	// Send Port
	ReconnectTimer		   : TON;
	ClientServerConnection : FB_ClientServerConnection;
	_ServerConnectionState : E_SocketConnectionState;
	SocketSend			   : FB_SocketSend;
	SendMessage			   : ST_TcpIpPayload;
	_Socket				   : T_HSOCKET;
	SendDelay			   : TON;
	PollTimer			   : TON;
	ResponseTimer		   : TON;
	SocketReceive		   : FB_SocketReceive;
	ReceiveMessage		   : ST_TcpIpPayload;

	//
	_ReconnectionTime : TIME := T#10S;
	_PollTime		  : TIME := T#100MS;
	_ReceiveTimeout	  : TIME := T#50S;
	_SendInterval	  : TIME := T#100MS;
END_VAR

VAR
	Commands		   : ARRAY[0..COMMAND_BUFFER] OF I_TcpIpSubscription;
	SendBuffer		   : ARRAY[0..COMMAND_BUFFER] OF ST_TcpIpPayload;
	PrioritySendBuffer : ARRAY[0..COMMAND_BUFFER] OF ST_TcpIpPayload;
END_VAR

VAR CONSTANT
	COMMAND_BUFFER : DINT := 99;
END_VAR

METHOD CyclicLogic
IF NOT _Initialized THEN
	Initialize();
	RETURN;
END_IF

SendReceiveSequence();
END_METHOD

METHOD Initialize
SocketCloseAll(sSrvNetId := '', bExecute := TRUE);
IF NOT SocketCloseAll.bBusy AND NOT SocketCloseAll.bError THEN
	_Initialized := TRUE;
END_IF
END_METHOD

{attribute 'monitoring' := 'call'}
PROPERTY Initialized : BOOL
GET
Initialized := _Initialized;
END_GET
SET
_Initialized := Initialized;
END_SET
END_PROPERTY

METHOD PROTECTED EvaluateResponse
VAR
	i : DINT;
END_VAR
FOR i := 0 TO COMMAND_BUFFER DO
	IF Commands[i] = 0 THEN
		EXIT;
	END_IF

	Commands[i].UpdateCommandResult(ADR(ReceiveMessage));
END_FOR

MEMSET(ADR(ReceiveMessage), 0, SIZEOF(ReceiveMessage));
END_METHOD

METHOD PROTECTED GetNextCommand
VAR
	i : DINT;
END_VAR
IF SendBuffer[0].Size <> 0 THEN
	MEMCPY(ADR(SendMessage), ADR(SendBuffer[0]), SIZEOF(SendBuffer[0]));
	FOR i := 0 TO (COMMAND_BUFFER - 1) DO
		MEMCPY(ADR(SendBuffer[i]), ADR(SendBuffer[i + 1]), SIZEOF(SendBuffer[i]));
	END_FOR
END_IF
END_METHOD

METHOD PROTECTED GetNextPriorityCommand
VAR
	i : DINT;
END_VAR
IF PrioritySendBuffer[0].Size <> 0 THEN
	MEMCPY(ADR(SendMessage), ADR(PrioritySendBuffer[0]), SIZEOF(PrioritySendBuffer[0]));
	FOR i := 0 TO (COMMAND_BUFFER - 1) DO
		MEMCPY(ADR(PrioritySendBuffer[i]), ADR(PrioritySendBuffer[i + 1]), SIZEOF(PrioritySendBuffer[i]));
	END_FOR
END_IF
END_METHOD

METHOD PROTECTED SendReceiveSequence
VAR_INST
	SequenceState : UDINT;
END_VAR
ClientServerConnection(sSrvNetID   := '',
					   sRemoteHost := _IP,
					   nRemotePort := _Port,
					   hSocket	   => _Socket,
					   eState	   => _ServerConnectionState);

SocketSend(sSrvNetId := '',
		   hSocket	 := _Socket,
		   cbLen	 := SendMessage.Size,
		   pSrc		 := ADR(SendMessage.Data),
		   tTimeout	 := T#5S);

SocketReceive(sSrvNetId := '',
			  hSocket	:= _Socket,
			  cbLen		:= SIZEOF(ReceiveMessage.Data),
			  pDest		:= ADR(ReceiveMessage.Data),
			  tTimeout	:= _ReceiveTimeout);

ReceiveMessage.Size := SIZEOF(ReceiveMessage.Data);

//
ReconnectTimer(PT := _ReconnectionTime);
PollTimer(PT := _PollTime);
ResponseTimer(PT := _ReceiveTimeout);
CASE SequenceState OF
	0:
		ClientServerConnection.bEnable := TRUE;
		IF _ServerConnectionState = eSOCKET_CONNECTED THEN
			SequenceState := SequenceState + 10;
		END_IF

		IF ClientServerConnection.bError THEN
			Trace.Error(_Name, CONCAT('ClientServerConnection.bError: ', TO_STRING(ClientServerConnection.nErrId)));
			SequenceState := 200;
		END_IF

	10:
		// SENDING -----------------------------------------------------------------------------------
		SendDelay(IN := NOT SendDelay.Q, PT := _SendInterval);
		IF SendMessage.Size = 0 THEN
			GetNextPriorityCommand();
		END_IF

		IF SendMessage.Size = 0 THEN
			GetNextCommand();
		END_IF

		IF SocketSend.bExecute AND NOT SocketSend.bBusy AND NOT SocketSend.bError THEN
			Trace.Info(_Name, 'Client sent');
			MEMSET(ADR(SendMessage), 0, SIZEOF(SendMessage));
			SocketSend.bExecute := FALSE;
		END_IF

		IF SendMessage.Size <> 0 AND NOT SocketSend.bExecute AND SendDelay.Q THEN
			SocketSend.bExecute := TRUE;
		END_IF

		IF SocketSend.bError THEN
			Trace.Error(_Name, CONCAT('SocketSend.bError: ', TO_STRING(SocketSend.nErrId)));
			SequenceState := 200;
		END_IF

		// RECEIVING -----------------------------------------------------------------------------------
		PollTimer.IN		   := TRUE;
		SocketReceive.bExecute := TRUE;
		IF PollTimer.Q AND NOT SocketReceive.bError AND NOT SocketReceive.bBusy THEN
			IF SocketReceive.nRecBytes > 0 THEN
				ResponseTimer.IN := FALSE;
				Trace.Info(_Name, 'Client recieved');
				EvaluateResponse();
			END_IF

			SequenceState := 11;
			// Stale connection, disconnected while socket was open
			IF SocketReceive.nRecBytes = 0 THEN
				ResponseTimer.IN := TRUE;
				IF ResponseTimer.Q THEN
					Trace.Error(_Name, 'Receive Connection stale - re-connect!');
					SequenceState := 200;
				END_IF
			END_IF
		END_IF

		IF SocketReceive.bError THEN
			Trace.Error(_Name, CONCAT('SocketReceive.bError: ', TO_STRING(SocketReceive.nErrId)));
			SequenceState := 200;
		END_IF

	11:
		PollTimer.IN		   := FALSE;
		SocketReceive.bExecute := FALSE;
		SequenceState		   := 10;

	200:
		ReconnectTimer.IN			   := TRUE;
		ResponseTimer.IN			   := FALSE;
		ClientServerConnection.bEnable := FALSE;
		SocketReceive.bExecute		   := FALSE;
		SocketSend.bExecute			   := FALSE;
		IF _ServerConnectionState = eSOCKET_DISCONNECTED AND ReconnectTimer.Q THEN
			ReconnectTimer.IN := FALSE;
			SequenceState	  := 0;
		END_IF
END_CASE
END_METHOD

{attribute 'monitoring' := 'call'}
PROPERTY ConnectionState : E_SocketConnectionState
GET
ConnectionState := _ServerConnectionState;
END_GET
END_PROPERTY

{attribute 'monitoring' := 'call'}
PROPERTY IP : T_IPv4Addr
SET
_IP := IP;
END_SET
END_PROPERTY

{attribute 'monitoring' := 'call'}
PROPERTY PollTime : TIME
SET
_PollTime := PollTime;
END_SET
END_PROPERTY

{attribute 'monitoring' := 'call'}
PROPERTY Port : UDINT
SET
_Port := Port;
END_SET
END_PROPERTY

{attribute 'monitoring' := 'call'}
PROPERTY ReceiveTimeout : TIME
SET
_ReceiveTimeout := ReceiveTimeout;
END_SET
END_PROPERTY

{attribute 'monitoring' := 'call'}
PROPERTY ReconnectionTime : TIME
SET
_ReconnectionTime := ReconnectionTime;
END_SET
END_PROPERTY

METHOD RegisterCommand
VAR_INPUT
	Command : I_TcpIpSubscription;
END_VAR

VAR
	i : DINT;
END_VAR
FOR i := 0 TO COMMAND_BUFFER DO
	IF Commands[i] = 0 THEN
		Commands[i] := Command;
		RETURN;
	END_IF
END_FOR
END_METHOD

METHOD SendCommand
VAR_INPUT
	Command : POINTER TO ST_TcpIpPayload;
END_VAR

VAR
	i : DINT;
END_VAR
FOR i := 0 TO COMMAND_BUFFER DO
	IF SendBuffer[i].Size = 0 THEN
		MEMCPY(ADR(SendBuffer[i]), Command, SIZEOF(SendBuffer[i]));
		RETURN;
	END_IF
END_FOR
END_METHOD

{attribute 'monitoring' := 'call'}
PROPERTY SendInterval : TIME
SET
_SendInterval := SendInterval;
END_SET
END_PROPERTY

METHOD SendPriorityCommand
VAR_INPUT
	Command : POINTER TO ST_TcpIpPayload;
END_VAR

VAR
	i : DINT;
END_VAR
FOR i := 0 TO COMMAND_BUFFER DO
	IF PrioritySendBuffer[i].Size = 0 THEN
		MEMCPY(ADR(PrioritySendBuffer[i]), Command, SIZEOF(PrioritySendBuffer[i]));
		RETURN;
	END_IF
END_FOR
END_METHOD

PROPERTY Socket : T_HSOCKET
GET
Socket := _Socket;
END_GET
END_PROPERTY

END_FUNCTION_BLOCK

// HMI/Interface/I_Button
INTERFACE I_Button EXTENDS I_Base

{attribute 'monitoring' := 'call'}
PROPERTY Active : BOOL
GET
END_GET
END_PROPERTY

{attribute 'monitoring' := 'call'}
PROPERTY Name : STRING
GET
END_GET
SET
END_SET
END_PROPERTY

PROPERTY Permissive : I_Permissive
GET
END_GET
END_PROPERTY

END_INTERFACE

// HMI/Interface/I_StringCollection
INTERFACE I_StringCollection

METHOD AddString
VAR_INPUT
	StringToAdd : T_MaxString;
END_VAR
END_METHOD

METHOD Clear : BOOL
VAR_INPUT
END_VAR
END_METHOD

PROPERTY Entries : UDINT
GET
END_GET
END_PROPERTY

END_INTERFACE

// HMI/Button
FUNCTION_BLOCK Button IMPLEMENTS I_Button
VAR
	_Name		: STRING;
	_Active		: BOOL;
	_Permissive : PermissiveInterlock;
END_VAR

{attribute 'monitoring' := 'call'}
PROPERTY Active : BOOL
GET
Active := _Active;
END_GET
END_PROPERTY

{attribute 'monitoring' := 'call'}
PROPERTY Name : STRING
GET
Name := _Name;
END_GET
SET
_Name := Name;
END_SET
END_PROPERTY

PROPERTY Permissive : I_Permissive
GET
Permissive := _Permissive;
END_GET
END_PROPERTY

END_FUNCTION_BLOCK

// Permissive Interlock/PermissiveInterlock
FUNCTION_BLOCK PermissiveInterlock IMPLEMENTS I_Permissive
VAR
	_OK				 : BOOL				   := TRUE;
	Permissive		 : ARRAY[0..9] OF BOOL := [TRUE, TRUE, TRUE, TRUE, TRUE, TRUE, TRUE, TRUE, TRUE, TRUE];
	PermissiveReason : ARRAY[0..9] OF STRING;
END_VAR

METHOD PROTECTED Check : BOOL
VAR
	i : UDINT;
END_VAR
_OK := TRUE;
FOR i := 0 TO 9 DO
	IF NOT Permissive[i] THEN
		_OK := FALSE;
	END_IF
END_FOR
END_METHOD

{attribute 'monitoring' := 'call'}
PROPERTY OK : BOOL
GET
OK := _OK;
END_GET
END_PROPERTY

METHOD Set
VAR_INPUT
	Index  : UDINT(0..9);
	Reason : STRING;
	Value  : BOOL;
END_VAR
Permissive[Index]		:= Value;
PermissiveReason[Index] := Reason;
Check();
END_METHOD

END_FUNCTION_BLOCK

// Kinematic Group/Interface/I_KinematicGroup
INTERFACE I_KinematicGroup EXTENDS I_Component, I_Override, I_TaskResult, I_Resettable

METHOD AddAcsAxis : BOOL
VAR_INPUT
	AxisId : UDINT;
END_VAR
END_METHOD

METHOD AddMcsAxis : BOOL
VAR_INPUT
	AxisId : UDINT;
END_VAR
END_METHOD

METHOD BuildGroup
VAR_INPUT
END_VAR
END_METHOD

METHOD DissolveGroup
VAR_INPUT
END_VAR
END_METHOD

{attribute 'monitoring' := 'call'}
PROPERTY Status : E_KinStatus
GET
END_GET
END_PROPERTY

END_INTERFACE

// Kinematic Group/KinematicGroup
FUNCTION_BLOCK KinematicGroup EXTENDS CyclicComponent IMPLEMENTS I_KinematicGroup, I_Initializable
VAR
	NcToPlc AT %I* : NCTOPLC_NCICHANNEL_REF;
	PlcToNc AT %Q* : PLCTONC_NCICHANNEL_REF;
	KinAxes		   : ST_KinAxes;
	KinConfigGroup : FB_KinConfigGroup;
	KinResetGroup  : FB_KinResetGroup;
	{attribute 'hide'}
	_Initialized : BOOL;
	{attribute 'hide'}
	_Busy : BOOL;
	{attribute 'hide'}
	_Error : BOOL;
	{attribute 'hide'}
	_ErrorId : UDINT;
END_VAR

METHOD DeregisterWithParent
VAR_INPUT
	Parent : I_ContainComponents;
END_VAR
SUPER^.DeregisterWithParent(Parent);
Parent.DeregisterInitialize(THIS^);
END_METHOD

METHOD RegisterWithParent
VAR_INPUT
	Parent : I_ContainComponents;
END_VAR
SUPER^.RegisterWithParent(Parent);
Parent.RegisterInitialize(THIS^);
END_METHOD

METHOD CyclicLogic
IF NOT Initialized THEN
	Initialize();
	RETURN;
END_IF

//
KinConfigGroup(stAxesList := KinAxes, stKinRefIn := NcToPlc);
IF KinConfigGroup.bError THEN
	_Error	 := TRUE;
	_ErrorId := KinConfigGroup.nErrorId;
END_IF

KinConfigGroup.bExecute := FALSE;

//
KinResetGroup(nItpChannelId := NcToPlc.ChnId, stKinRefIn := NcToPlc, stAxesList := KinAxes);
IF KinResetGroup.bError THEN
	_Error	 := TRUE;
	_ErrorId := KinResetGroup.nErrorId;
END_IF

KinResetGroup.bExecute := FALSE;

//
_Busy := KinConfigGroup.bBusy;
END_METHOD

METHOD Initialize
VAR
	i : DINT;
END_VAR
IF NOT Initialized THEN
	IF KinAxes.nAxisIdsAcs[1] = 0 THEN
		Trace.LogMessage(Name, 'Init failed - at least one ACS Axis needs to be added to Kinematic!');
		RETURN;
	END_IF

	IF KinAxes.nAxisIdsMcs[1] = 0 THEN
		Trace.LogMessage(Name, 'Init failed - at least one MCS Axis needs to be added to Kinematic!');
		RETURN;
	END_IF

	IF F_GetMappingStatus(ADR(NcToPlc), SIZEOF(NcToPlc)) <> EPlcMappingStatus.MS_Mapped THEN
		Trace.LogMessage(Name, 'Init failed - NcToPlc not mapped to Kinematic Channel!');
		RETURN;
	END_IF

	IF F_GetMappingStatus(ADR(PlcToNc), SIZEOF(PlcToNc)) <> EPlcMappingStatus.MS_Mapped THEN
		Trace.LogMessage(Name, 'Init failed - PlcToNc not mapped to Kinematic Channel!');
		RETURN;
	END_IF

	Initialized := TRUE;
END_IF
END_METHOD

{attribute 'monitoring' := 'call'}
PROPERTY Initialized : BOOL
GET
Initialized := _Initialized;
END_GET
SET
_Initialized := Initialized;
END_SET
END_PROPERTY

METHOD AddAcsAxis : BOOL
VAR_INPUT
	AxisId : UDINT;
END_VAR

VAR
	i : DINT;
END_VAR
IF AxisId = 0 THEN
	RETURN;
END_IF

FOR i := 1 TO 8 DO
	IF KinAxes.nAxisIdsAcs[i] = 0 THEN
		KinAxes.nAxisIdsAcs[i] := AxisId;
		AddAcsAxis			   := TRUE;
		RETURN;
	END_IF
END_FOR
END_METHOD

METHOD AddMcsAxis : BOOL
VAR_INPUT
	AxisId : UDINT;
END_VAR

VAR
	i : DINT;
END_VAR
IF AxisId = 0 THEN
	RETURN;
END_IF

FOR i := 1 TO 8 DO
	IF KinAxes.nAxisIdsMcs[i] = 0 THEN
		KinAxes.nAxisIdsMcs[i] := AxisId;
		AddMcsAxis			   := TRUE;
		RETURN;
	END_IF
END_FOR
END_METHOD

METHOD BuildGroup
VAR_INPUT
END_VAR
IF Busy THEN
	RETURN;
END_IF

KinConfigGroup.bCartesianMode := TRUE;
KinConfigGroup.bExecute		  := TRUE;
END_METHOD

METHOD DissolveGroup
VAR_INPUT
END_VAR
IF Busy THEN
	RETURN;
END_IF

KinConfigGroup.bCartesianMode := FALSE;
KinConfigGroup.bExecute		  := TRUE;
END_METHOD

{attribute 'monitoring' := 'call'}
PROPERTY Override : LREAL
SET
PlcToNc.ChnAxesOvr	  := TO_UDINT(Override * 10_000);
PlcToNc.ChnSpindleOvr := TO_UDINT(Override * 10_000);
END_SET
END_PROPERTY

{attribute 'monitoring' := 'call'}
PROPERTY Status : E_KinStatus
GET
Status := F_KinGetChnOperationState(NcToPlc);
END_GET
END_PROPERTY

METHOD Reset
_Error				   := FALSE;
_ErrorId			   := 0;
KinResetGroup.bExecute := TRUE;
END_METHOD

{attribute 'monitoring' := 'call'}
PROPERTY Busy : BOOL
GET
Busy := _Busy;
END_GET
END_PROPERTY

{attribute 'monitoring' := 'call'}
PROPERTY Error : BOOL
GET
Error := _Error;
END_GET
END_PROPERTY

{attribute 'monitoring' := 'call'}
PROPERTY ErrorId : UDINT
GET
ErrorId := _ErrorId;
END_GET
END_PROPERTY

END_FUNCTION_BLOCK

// Kinematic Group/KinematicGroup_TcEvents
FUNCTION_BLOCK KinematicGroup_TcEvents EXTENDS CyclicComponent IMPLEMENTS I_EventReactionTcEvents
VAR
	KinematicGroup : I_KinematicGroup;
	Events		   : TcEventClass('Kinematic Group Events');
END_VAR

METHOD GetHighestActiveEventReaction : DINT
GetHighestActiveEventReaction := Events.GetHighestActiveEventReaction();
END_METHOD

METHOD GetHighestActiveEventSeverity : TcEventSeverity
GetHighestActiveEventSeverity := Events.GetHighestActiveEventSeverity();
END_METHOD

METHOD Reset
Events.Reset();
END_METHOD

METHOD SetEventReactions
VAR_INPUT
	Verbose	 : DINT := 0;
	Info	 : DINT := 1;
	Warning	 : DINT := 2;
	Error	 : DINT := 3;
	Critical : DINT := 4;
END_VAR
Events.SetEventReactions(Verbose,
						 Info,
						 Warning,
						 Error,
						 Critical);
END_METHOD

METHOD CyclicLogic
IF KinematicGroup = 0 THEN
	RETURN;
END_IF

IF KinematicGroup.Error THEN
	Events.Arguments(E_KinematicGroup.KinematicGroupError).Clear().AddString(TO_STRING(KinematicGroup.ErrorId));
	Events.RaiseEvent(E_KinematicGroup.KinematicGroupError);
END_IF
END_METHOD

(*FB_Init is always available implicitly and it is used primarily for initialization.
The return value is not evaluated. For a specific influence, you can also declare the
methods explicitly and provide additional code there with the standard initialization
code. You can evaluate the return value.*)
METHOD FB_Init : BOOL
VAR_INPUT
	(* TRUE: the retain variables are initialized (reset warm / reset cold)*)
	bInitRetains : BOOL;

	(* TRUE: the instance will be copied to the copy code afterward (online change)   *)
	bInCopyCode	   : BOOL;
	Name		   : T_MaxString;
	KinematicGroup : I_KinematicGroup;
END_VAR
THIS^.KinematicGroup := KinematicGroup;
Events.GenerateTcEvents(KinematicGroup.Name, ADR(TC_Events.KinematicGroup), SIZEOF(ST_KinematicGroup));
END_METHOD

END_FUNCTION_BLOCK

// Modes/PackMLModeControl
FUNCTION_BLOCK PackMLModeControl IMPLEMENTS I_Mode, I_Cyclic
VAR
	{attribute 'hide'}
	_CurrentMode : DINT;
	{attribute 'hide'}
	ModeManager	  : FB_PMLUnitModeManager;
	ModeCommand	  : DINT;
	_StateMachine : I_Statemachine;
END_VAR

METHOD ChangeMode
VAR_INPUT
	RequestedMode : DINT;
END_VAR
IF RequestedMode <= 0 OR RequestedMode > 31 THEN
	Trace.LogMessage('PackML Mode Controller', ' - Requested Mode is not valid 1..31');
	RETURN;
END_IF

ModeCommand := RequestedMode;
END_METHOD

{attribute 'monitoring' := 'call'}
PROPERTY CurrentMode : DINT
GET
CurrentMode := _CurrentMode;
END_GET
END_PROPERTY

METHOD CyclicLogic
VAR_INST
	LastModeCommand		: DINT;
	ModeChangeRequested : BOOL;
END_VAR
IF _CurrentMode = 0 THEN
	ModeChangeRequested := TRUE;
	ModeCommand			:= E_PMLProtectedUnitMode.Production;
	LastModeCommand		:= ModeCommand;
ELSIF ModeCommand <> LastModeCommand THEN
	ModeChangeRequested := TRUE;
	LastModeCommand		:= ModeCommand;
END_IF

IF ModeChangeRequested THEN
	{warning disable C0196}
	ModeManager(bExecute	 := TRUE,
				eModeCommand := ModeCommand,
				eState		 := _StateMachine.CurrentState,
				eModeStatus	 => _CurrentMode);

	IF ModeManager.bDone THEN
		ModeManager(bExecute := FALSE);
		ModeChangeRequested := FALSE;
	ELSIF ModeManager.bError THEN
		IF ModeManager.nErrorId = 1 THEN
			Trace.LogMessage('PackML Mode Controller', 'Requested mode is not defined or Mode change is disabled in this PackML state!');
		ELSE
			Trace.LogMessage('PackML Mode Controller', 'Mode change error, check PackML configuration!');
		END_IF

		ModeManager(bExecute := FALSE);
		_StateMachine.ChangeState(TO_UDINT(E_PMLCommand.Abort));
		ModeCommand			:= E_PMLProtectedUnitMode.Production;
		ModeChangeRequested := FALSE;
	END_IF
END_IF
END_METHOD

PROPERTY StateMachine : I_StateMachine
SET
_StateMachine := StateMachine;
END_SET
END_PROPERTY

END_FUNCTION_BLOCK

// Module PackML/PackMLModule
FUNCTION_BLOCK ABSTRACT PackMLModule EXTENDS Module IMPLEMENTS I_Module, I_ContainStatemachine
VAR
	_Statemachine : PackMLStatemachine_ModuleIntegrated('Statemachine');
	SequenceState : UDINT;
END_VAR

(*FB_Init is always available implicitly and it is used primarily for initialization.
The return value is not evaluated. For a specific influence, you can also declare the
methods explicitly and provide additional code there with the standard initialization
code. You can evaluate the return value.*)
METHOD FB_Init : BOOL
VAR_INPUT
	(* TRUE: the retain variables are initialized (reset warm / reset cold)*)
	bInitRetains	: BOOL;
	(* TRUE: the instance will be copied to the copy code afterward (online change)   *)
	bInCopyCode	: BOOL;
	Name	: T_MaxString;
END_VAR
_Statemachine.RegisterWithParent(THIS^);
END_METHOD

METHOD Aborted : BOOL;
Aborted := TRUE;
END_METHOD

METHOD Aborting : BOOL
Aborting := TRUE;
END_METHOD

METHOD Clearing : BOOL
Clearing := TRUE;
END_METHOD

METHOD Completed : BOOL
Completed := TRUE;
END_METHOD

METHOD Completing : BOOL
Completing := TRUE;
END_METHOD

METHOD Execute : BOOL
Execute := TRUE;
END_METHOD

METHOD Held : BOOL
Held := TRUE;
END_METHOD

METHOD Holding : BOOL
Holding := TRUE;
END_METHOD

METHOD Idle : BOOL
Idle := TRUE;
END_METHOD

METHOD Resetting : BOOL
Resetting := TRUE;
END_METHOD

METHOD Starting : BOOL
Starting := TRUE;
END_METHOD

METHOD Stopped : BOOL
Stopped := TRUE;
END_METHOD

METHOD Stopping : BOOL
Stopping := TRUE;
END_METHOD

METHOD Suspended : BOOL
Suspended := TRUE;
END_METHOD

METHOD Suspending : BOOL
Suspending := TRUE;
END_METHOD

METHOD Unholding : BOOL
Unholding := TRUE;
END_METHOD

METHOD Unsuspending : BOOL
Unsuspending := TRUE;
END_METHOD

METHOD CyclicLogic
StateSelect();
SUPER^.CyclicLogic();
END_METHOD

PROPERTY Statemachine : I_Statemachine
GET
Statemachine := _Statemachine;
END_GET
END_PROPERTY

METHOD PRIVATE StateSelect
VAR_INST
	ClearingTon : TON;
	LastState	: DINT;
END_VAR
IF LastState <> _Statemachine.CurrentState THEN
	SequenceState := 0;
	LastState	  := _Statemachine.CurrentState;
END_IF

CASE _Statemachine.CurrentState OF
	E_PMLState.Undefined:
		;

	E_PMLState.Clearing:
		ClearingTon(IN := TRUE, PT := ApplicationBaseParameter.ClearingTimeout);
		IF Clearing() THEN
			ClearingTon(IN := FALSE);
			_Statemachine.StateComplete();
		END_IF

		IF ClearingTon.Q THEN
			ClearingTon(IN := FALSE);
			Trace.LogMessage('Clearing Timeout exeeded! - ', _Name);
			_Statemachine.ChangeState(E_PMLCommand.Abort);
		END_IF

	E_PMLState.Stopped:
		Stopped();

	E_PMLState.Starting:
		IF Starting() THEN
			_Statemachine.StateComplete();
		END_IF

	E_PMLState.Idle:
		Idle();

	E_PMLState.Suspended:
		Suspended();

	E_PMLState.Execute:
		Execute();

	E_PMLState.Stopping:
		IF Stopping() THEN
			_Statemachine.StateComplete();
		END_IF

	E_PMLState.Aborting:
		IF Aborting() THEN
			_Statemachine.StateComplete();
		END_IF

	E_PMLState.Aborted:
		Aborted();

	E_PMLState.Holding:
		IF Holding() THEN
			_Statemachine.StateComplete();
		END_IF

	E_PMLState.Held:
		Held();

	E_PMLState.Unholding:
		IF Unholding() THEN
			_Statemachine.StateComplete();
		END_IF

	E_PMLState.Suspending:
		IF Suspending() THEN
			_Statemachine.StateComplete();
		END_IF

	E_PMLState.Unsuspending:
		IF Unsuspending() THEN
			_Statemachine.StateComplete();
		END_IF

	E_PMLState.Resetting:
		IF Resetting() THEN
			_Statemachine.StateComplete();
		END_IF

	E_PMLState.Completing:
		IF Completing() THEN
			_Statemachine.StateComplete();
		END_IF

	E_PMLState.Completed:
		Completed();
END_CASE
END_METHOD

END_FUNCTION_BLOCK

// Statemachine/Interface/I_ContainStatemachine
INTERFACE I_ContainStatemachine EXTENDS I_Base

PROPERTY Statemachine : I_Statemachine
GET
END_GET
END_PROPERTY

END_INTERFACE

// Statemachine/PackML/PackMLStatemachine_ModuleIntegrated
FUNCTION_BLOCK PackMLStatemachine_ModuleIntegrated EXTENDS CyclicComponent IMPLEMENTS I_StateMachine
VAR
	StateMachine   : FB_PMLStateMachine;
	StateCommand   : E_PMLCommand;
	_CurrentState  : E_PMLState;
	ModeController : PackMLModeControl := (StateMachine := THIS^);
END_VAR

PROPERTY Mode : I_Mode
GET
Mode := ModeController;
END_GET
SET
// Fix defined in PackML
END_SET
END_PROPERTY

METHOD ChangeState
VAR_INPUT
	StateCommand : DINT;
END_VAR
IF StateCommand <= 0 OR StateCommand > 17 THEN
	Trace.LogMessage('PackML Statemachine ChangeState()', 'StateId is not a PackML State');
END_IF

{warning disable C0196}
THIS^.StateCommand := StateCommand;
END_METHOD

{attribute 'monitoring' := 'call'}
PROPERTY CurrentState : DINT
GET
CurrentState := _CurrentState;
END_GET
END_PROPERTY

METHOD CyclicLogic
VAR_INST
	ClearingTon : TON;
END_VAR
ModeController.CyclicLogic();
IF _CurrentState = E_PMLState.Undefined AND Mode.CurrentMode <> 0 THEN
	StateCommand := E_PMLCommand.Abort;
END_IF

StateMachine(eMode			  := TO_DINT(Mode.CurrentMode),
			 eCommand		  := StateCommand,
			 stSubUnitInfoRef :=,
			 stOptions		  :=,
			 eState			  => _CurrentState,
			 sState			  =>,
			 bError			  =>,
			 nErrorID		  =>);

CASE _CurrentState OF
	E_PMLState.Clearing:
		ClearingTon(IN := TRUE, PT := ApplicationBaseParameter.ClearingTimeout);
		IF ClearingTon.Q THEN
			ClearingTon(IN := FALSE);
			Trace.LogMessage('Clearing Timeout exeeded!', 'ApplicationBaseParameter.ClearingTimeout');
			StateCommand := E_PMLCommand.Abort;
		END_IF

ELSE
	ClearingTon(IN := FALSE);
END_CASE
END_METHOD

METHOD StateComplete
StateMachine.M_StateComplete();
END_METHOD

{attribute 'hide'} 
PROPERTY States : I_StateList
GET
States := 0;
END_GET
END_PROPERTY

END_FUNCTION_BLOCK

// Motion/Interface/I_Axis_PTP
INTERFACE I_Axis_PTP EXTENDS I_Axis, I_AxisMoveAbsolute, I_AxisMoveModulo, I_AxisMoveRelative, I_AxisMoveVelocity

END_INTERFACE

// Motion/Interface/I_AxisMoveAbsolute
INTERFACE I_AxisMoveAbsolute EXTENDS I_Base

METHOD MoveAbsolute
VAR_INPUT
	TargetPosition : LREAL;
	AbortPrevious  : BOOL := TRUE;
END_VAR
END_METHOD

END_INTERFACE

// Motion/Interface/I_AxisMoveModulo
INTERFACE I_AxisMoveModulo EXTENDS I_Base

METHOD MoveModulo : BOOL
VAR_INPUT
	Position	  : LREAL;
	Direction	  : MC_Direction := MC_Direction.MC_Shortest_Way;
	AbortPrevious : BOOL		 := TRUE;
END_VAR
END_METHOD

END_INTERFACE

// Motion/Interface/I_AxisMoveRelative
INTERFACE I_AxisMoveRelative EXTENDS I_Base

METHOD MoveRelative : BOOL
VAR_INPUT
	Distance	  : LREAL;
	AbortPrevious : BOOL := TRUE;
END_VAR
END_METHOD

END_INTERFACE

// Motion/Interface/I_AxisMoveVelocity
INTERFACE I_AxisMoveVelocity EXTENDS I_Base

METHOD MoveVelocity : BOOL
VAR_INPUT
	Velocity	  : LREAL;
	AbortPrevious : BOOL := TRUE;
END_VAR
END_METHOD

END_INTERFACE

// Motion/Interface/I_AxisGear
INTERFACE I_AxisGear EXTENDS I_Base

METHOD GearIn
VAR_INPUT
END_VAR
END_METHOD

PROPERTY GearInMultiMasterOptions : ST_GearInMultiMasterOptions
SET
END_SET
END_PROPERTY

METHOD GearOut
VAR_INPUT
END_VAR
END_METHOD

{attribute 'monitoring' := 'call'}
PROPERTY GearRatioMaster1 : LREAL
SET
END_SET
END_PROPERTY

{attribute 'monitoring' := 'call'}
PROPERTY GearRatioMaster2 : LREAL
SET
END_SET
END_PROPERTY

{attribute 'monitoring' := 'call'}
PROPERTY GearRatioMaster3 : LREAL
SET
END_SET
END_PROPERTY

{attribute 'monitoring' := 'call'}
PROPERTY GearRatioMaster4 : LREAL
SET
END_SET
END_PROPERTY

PROPERTY Master1 : I_Axis
SET
END_SET
END_PROPERTY

PROPERTY Master2 : I_Axis
SET
END_SET
END_PROPERTY

PROPERTY Master3 : I_Axis
SET
END_SET
END_PROPERTY

PROPERTY Master4 : I_Axis
SET
END_SET
END_PROPERTY

END_INTERFACE

// Motion/Interface/I_SlaveAxis
INTERFACE I_SlaveAxis EXTENDS I_Axis_PTP, I_AxisGear

END_INTERFACE

// Motion/Axis_TcEvents
FUNCTION_BLOCK Axis_TcEvents EXTENDS CyclicComponent IMPLEMENTS I_EventReactionTcEvents
VAR
	Axis   : I_Axis;
	Events : TcEventClass(CONCAT(Name, ' Events'));
END_VAR

METHOD GetHighestActiveEventReaction : DINT
GetHighestActiveEventReaction := Events.GetHighestActiveEventReaction();
END_METHOD

METHOD GetHighestActiveEventSeverity : TcEventSeverity
GetHighestActiveEventSeverity := Events.GetHighestActiveEventSeverity();
END_METHOD

METHOD Reset
Events.Reset();
END_METHOD

METHOD SetEventReactions
VAR_INPUT
	Verbose	 : DINT := 0;
	Info	 : DINT := 1;
	Warning	 : DINT := 2;
	Error	 : DINT := 3;
	Critical : DINT := 4;
END_VAR
Events.SetEventReactions(Verbose,
						 Info,
						 Warning,
						 Error,
						 Critical);
END_METHOD

METHOD CyclicLogic
IF Axis.MotionTasks.Error THEN
	Events.Arguments(E_Nc2Axis.AxisError).Clear().AddString(Axis.MotionTasks.ErrorTask).AddString(TO_STRING(Axis.MotionTasks.ErrorId));
	Events.RaiseEvent(E_Nc2Axis.AxisError);
END_IF
END_METHOD

(*FB_Init is always available implicitly and it is used primarily for initialization.
The return value is not evaluated. For a specific influence, you can also declare the
methods explicitly and provide additional code there with the standard initialization
code. You can evaluate the return value.*)
METHOD FB_Init : BOOL
VAR_INPUT
	(* TRUE: the retain variables are initialized (reset warm / reset cold)*)
	bInitRetains : BOOL;

	(* TRUE: the instance will be copied to the copy code afterward (online change)   *)
	bInCopyCode : BOOL;
	Name		: T_MaxString;
	Axis		: I_Axis;
END_VAR
THIS^.Axis := Axis;
Events.GenerateTcEvents(Axis.Name, ADR(TC_events.Nc2Axis), SIZEOF(ST_Nc2Axis));
END_METHOD

END_FUNCTION_BLOCK

// Motion/AxisPTP
FUNCTION_BLOCK AxisPTP EXTENDS Axis IMPLEMENTS I_Axis_PTP
VAR
	// Tasks
	{attribute 'hide'}
	MoveAbsoluteTask : MoveAbsoluteTask := (Name := 'MC Move Absolute');
	{attribute 'hide'}
	MoveRelativeTask : MoveRelativeTask := (Name := 'MC Move Relative');
	{attribute 'hide'}
	MoveModuloTask : MoveModuloTask := (Name := 'MC Move Modulo');
	{attribute 'hide'}
	MoveVelocityTask : MoveVelocityTask := (Name := 'MC Move Velocity');
END_VAR

(*FB_Init is always available implicitly and it is used primarily for initialization.
The return value is not evaluated. For a specific influence, you can also declare the
methods explicitly and provide additional code there with the standard initialization
code. You can evaluate the return value.*)
METHOD FB_Init : BOOL
VAR_INPUT
	(* TRUE: the retain variables are initialized (reset warm / reset cold)*)
	bInitRetains : BOOL;

	(* TRUE: the instance will be copied to the copy code afterward (online change)   *)
	bInCopyCode : BOOL;
	Name		: T_MaxString;
	Axis		: REFERENCE TO AXIS_REF;
END_VAR
// Register all Motion Tasks to Collection
MotionTaskCollection.AddTask(MoveAbsoluteTask);
MotionTaskCollection.AddTask(MoveRelativeTask);
MotionTaskCollection.AddTask(MoveModuloTask);
MotionTaskCollection.AddTask(MoveVelocityTask);
END_METHOD

METHOD MoveAbsolute
VAR_INPUT
	TargetPosition : LREAL;
	AbortPrevious  : BOOL := TRUE;
END_VAR
IF Error THEN
	RETURN;
ELSE
	IF Busy AND NOT AbortPrevious THEN
		RETURN;
	END_IF
END_IF

MoveAbsoluteTask.BufferMode		:= _McBufferMode;
MoveAbsoluteTask.MoveOptions	:= _MoveOptions;
MoveAbsoluteTask.TargetPosition := TargetPosition;
MoveAbsoluteTask.Execute();
END_METHOD

METHOD MoveModulo : BOOL
VAR_INPUT
	Position	: LREAL;
	Direction	: MC_Direction := .MC_Direction.MC_Shortest_Way;
	AbortPrevious	: BOOL := TRUE;
END_VAR
IF Error THEN
	RETURN;
ELSE
	IF Busy AND NOT AbortPrevious THEN
		RETURN;
	END_IF
END_IF

MoveModuloTask.BufferMode	  := _McBufferMode;
MoveModuloTask.MoveOptions	  := _MoveOptions;
MoveModuloTask.Direction	  := Direction;
MoveModuloTask.TargetPosition := Position;
MoveModuloTask.Execute();
END_METHOD

METHOD MoveRelative : BOOL
VAR_INPUT
	Distance	  : LREAL;
	AbortPrevious : BOOL := TRUE;
END_VAR
IF Error THEN
	RETURN;
ELSE
	IF Busy AND NOT AbortPrevious THEN
		RETURN;
	END_IF
END_IF

MoveRelativeTask.BufferMode		:= _McBufferMode;
MoveRelativeTask.MoveOptions	:= _MoveOptions;
MoveRelativeTask.TargetDistance := Distance;
MoveRelativeTask.Execute();
END_METHOD

METHOD MoveVelocity : BOOL
VAR_INPUT
	Velocity	  : LREAL;
	AbortPrevious : BOOL := TRUE;
END_VAR
IF Error THEN
	RETURN;
ELSE
	IF Busy AND NOT AbortPrevious THEN
		RETURN;
	END_IF
END_IF

MoveVelocityTask.BufferMode		:= _McBufferMode;
MoveVelocityTask.MoveOptions	:= _MoveOptions;
MoveVelocityTask.TargetVelocity := Velocity;
MoveVelocityTask.Execute();
END_METHOD

END_FUNCTION_BLOCK

// Motion/AxisPTP_HMI
FUNCTION_BLOCK AxisPTP_HMI EXTENDS HmiFunction
VAR
	Axis : I_Axis_PTP;
	{ attribute 'TcHmiSymbol.AddSymbol' }
	{ attribute 'TcHmiSymbol.AddSymbol.UserGroups' := '__SystemAdministrators,Admin' }
	AxisPTP_HMI : ST_AxisPTP_HMI;
END_VAR

PROPERTY DisablePermissive : I_Permissive
GET
DisablePermissive := AxisPTP_HMI.Disable.Permissive;
END_GET
END_PROPERTY

PROPERTY EnablePermissive : I_Permissive
GET
EnablePermissive := AxisPTP_HMI.Enable.Permissive;
END_GET
END_PROPERTY

PROPERTY HomePermissive : I_Permissive
GET
HomePermissive := AxisPTP_HMI.Home.Permissive;
END_GET
END_PROPERTY

PROPERTY JogBackwardFastPermissive : I_Permissive
GET
JogBackwardFastPermissive := AxisPTP_HMI.JogBackwardFast.Permissive;
END_GET
END_PROPERTY

PROPERTY JogBackwardSlowPermissive : I_Permissive
GET
JogBackwardSlowPermissive := AxisPTP_HMI.JogBackwardSlow.Permissive;
END_GET
END_PROPERTY

PROPERTY JogForwardFastPermissive : I_Permissive
GET
JogForwardFastPermissive := AxisPTP_HMI.JogForwardFast.Permissive;
END_GET
END_PROPERTY

PROPERTY JogForwardSlowPermissive : I_Permissive
GET
JogForwardSlowPermissive := AxisPTP_HMI.JogForwardSlow.Permissive;
END_GET
END_PROPERTY

PROPERTY MoveAbsolutePermissive : I_Permissive
GET
MoveAbsolutePermissive := AxisPTP_HMI.MoveAbsolute.Permissive;
END_GET
END_PROPERTY

PROPERTY MoveModuloPermissive : I_Permissive
GET
MoveModuloPermissive := AxisPTP_HMI.MoveModulo.Permissive;
END_GET
END_PROPERTY

PROPERTY MoveRelativePermissive : I_Permissive
GET
MoveRelativePermissive := AxisPTP_HMI.MoveRelative.Permissive;
END_GET
END_PROPERTY

PROPERTY MoveVelocityPermissive : I_Permissive
GET
MoveVelocityPermissive := AxisPTP_HMI.MoveVelocity.Permissive;
END_GET
END_PROPERTY

PROPERTY ResetPermissive : I_Permissive
GET
ResetPermissive := AxisPTP_HMI.Reset.Permissive;
END_GET
END_PROPERTY

PROPERTY StopPermissive : I_Permissive
GET
StopPermissive := AxisPTP_HMI.Stop.Permissive;
END_GET
END_PROPERTY

PROPERTY ControlObject : I_Base
SET
__QueryInterface(ControlObject,Axis);
END_SET
END_PROPERTY

METHOD CyclicLogic
VAR_INST
	EnableRT	   : R_TRIG;
	DisableRT	   : R_TRIG;
	StopRT		   : R_TRIG;
	HomeRT		   : R_TRIG;
	ResetRT		   : R_TRIG;
	MoveAbsoluteRT : R_TRIG;
	MoveModuloRT   : R_TRIG;
	MoveRelativeRT : R_TRIG;
	MoveVelocityRT : R_TRIG;
END_VAR
IF Axis = 0 THEN
	RETURN;
END_IF

AxisPTP_HMI.HmiEnabled			 := Enabled;
AxisPTP_HMI.ActualAcceleration	 := Axis.ActualAcceleration;
AxisPTP_HMI.ActualPosition		 := Axis.ActualPosition;
AxisPTP_HMI.ActualPositionModulo := Axis.ActualPositionModulo;
AxisPTP_HMI.ActualTorque		 := Axis.ActualTorque;
AxisPTP_HMI.ActualVelocity		 := Axis.ActualVelocity;
AxisPTP_HMI.Busy				 := Axis.Busy;
AxisPTP_HMI.Error				 := Axis.Error;
AxisPTP_HMI.ErrorId				 := Axis.ErrorId;
AxisPTP_HMI.Name				 := Axis.Name;
AxisPTP_HMI.Status				 := Axis.Axis.Status;

// HMI Commands
StopRT(CLK := AxisPTP_HMI.Stop.Active);
IF StopRT.Q THEN
	IF AxisPTP_HMI.Stop.Permissive.OK THEN
		Axis.Stop();
	END_IF
END_IF

ResetRT(CLK := AxisPTP_HMI.Reset.Active);
IF ResetRT.Q THEN
	IF AxisPTP_HMI.Reset.Permissive.OK THEN
		Axis.Reset();
	END_IF
END_IF

IF Enabled THEN
	EnableRT(CLK := AxisPTP_HMI.Enable.Active);
	IF EnableRT.Q THEN
		IF AxisPTP_HMI.Enable.Permissive.OK THEN
			Axis.Enable();
		END_IF
	END_IF

	DisableRT(CLK := AxisPTP_HMI.Disable.Active);
	IF DisableRT.Q THEN
		IF AxisPTP_HMI.Disable.Permissive.OK THEN
			Axis.Disable();
		END_IF
	END_IF

	IF AxisPTP_HMI.JogBackwardSlow.Active THEN
		IF AxisPTP_HMI.JogBackwardSlow.Permissive.OK THEN
			Axis.Jog(JogForward := FALSE, JogBackwards := TRUE, JogMode := E_JogMode.MC_JOGMODE_STANDARD_SLOW);
		END_IF
	ELSIF AxisPTP_HMI.JogForwardSlow.Active THEN
		Axis.Jog(JogForward := TRUE, JogBackwards := FALSE, JogMode := E_JogMode.MC_JOGMODE_STANDARD_SLOW);
	ELSIF AxisPTP_HMI.JogBackwardFast.Active THEN
		Axis.Jog(JogForward := FALSE, JogBackwards := TRUE, JogMode := E_JogMode.MC_JOGMODE_STANDARD_FAST);
	ELSIF AxisPTP_HMI.JogForwardFast.Active THEN
		Axis.Jog(JogForward := TRUE, JogBackwards := FALSE, JogMode := E_JogMode.MC_JOGMODE_STANDARD_FAST);
	ELSE
		Axis.Jog(JogForward := FALSE, JogBackwards := FALSE, JogMode := E_JogMode.MC_JOGMODE_STANDARD_SLOW);
	END_IF

	HomeRT(CLK := AxisPTP_HMI.Home.Active);
	IF HomeRT.Q THEN
		IF AxisPTP_HMI.Home.Permissive.OK THEN
			Axis.Home();
		END_IF
	END_IF

	MoveAbsoluteRT(CLK := AxisPTP_HMI.MoveAbsolute.Active);
	IF MoveAbsoluteRT.Q THEN
		IF AxisPTP_HMI.MoveAbsolute.Permissive.OK THEN
			Axis.MoveAbsolute(AxisPTP_HMI.TargetPosition);
		END_IF
	END_IF

	MoveModuloRT(CLK := AxisPTP_HMI.MoveModulo.Active);
	IF MoveModuloRT.Q THEN
		IF AxisPTP_HMI.MoveModulo.Permissive.OK THEN
			Axis.MoveModulo(AxisPTP_HMI.TargetPosition);
		END_IF
	END_IF

	MoveRelativeRT(CLK := AxisPTP_HMI.MoveRelative.Active);
	IF MoveRelativeRT.Q THEN
		IF AxisPTP_HMI.MoveRelative.Permissive.OK THEN
			Axis.MoveRelative(AxisPTP_HMI.TargetDistance);
		END_IF
	END_IF

	MoveVelocityRT(CLK := AxisPTP_HMI.MoveVelocity.Active);
	IF MoveVelocityRT.Q THEN
		IF AxisPTP_HMI.MoveVelocity.Permissive.OK THEN
			Axis.MoveVelocity(AxisPTP_HMI.TargetVelocity);
		END_IF
	END_IF
END_IF
END_METHOD

(*FB_Init is always available implicitly and it is used primarily for initialization.
The return value is not evaluated. For a specific influence, you can also declare the
methods explicitly and provide additional code there with the standard initialization
code. You can evaluate the return value.*)
METHOD FB_Init : BOOL
VAR_INPUT
	(* TRUE: the retain variables are initialized (reset warm / reset cold)*)
	bInitRetains : BOOL;

	(* TRUE: the instance will be copied to the copy code afterward (online change)   *)
	bInCopyCode : BOOL;
	Name		: T_MaxString;
	Axis		: I_Axis_PTP;
	Unit		: STRING;
END_VAR
THIS^.Axis		 := Axis;
ControlType		 := 'AxisPTP';
LinkObject		 := 'AxisPTP_HMI';
AxisPTP_HMI.Unit := Unit;
END_METHOD

END_FUNCTION_BLOCK

// Motion/SlaveAxisPTP
FUNCTION_BLOCK SlaveAxisPTP EXTENDS AxisPTP IMPLEMENTS I_SlaveAxis
VAR
	// Tasks
	MotionCoupleTaskGearing : MotionCoupleTask_Gearing := (Name := 'MC GearIn Multimaster');
END_VAR

(*FB_Init is always available implicitly and it is used primarily for initialization.
The return value is not evaluated. For a specific influence, you can also declare the
methods explicitly and provide additional code there with the standard initialization
code. You can evaluate the return value.*)
METHOD FB_Init : BOOL
VAR_INPUT
	(* TRUE: the retain variables are initialized (reset warm / reset cold)*)
	bInitRetains : BOOL;

	(* TRUE: the instance will be copied to the copy code afterward (online change)   *)
	bInCopyCode : BOOL;
	Name		: T_MaxString;
	Axis		: REFERENCE TO AXIS_REF;
END_VAR
// Register all Motion Tasks to Collection
MotionTaskCollection.AddTask(MotionCoupleTaskGearing);
END_METHOD

METHOD GearIn
VAR_INPUT
END_VAR
MotionCoupleTaskGearing.GearIn	   := TRUE;
MotionCoupleTaskGearing.BufferMode := _McBufferMode;
MotionCoupleTaskGearing.Execute();
END_METHOD

PROPERTY GearInMultiMasterOptions : ST_GearInMultiMasterOptions
SET
MotionCoupleTaskGearing.GearInMultiMasterOptions := GearInMultiMasterOptions;
END_SET
END_PROPERTY

METHOD GearOut
VAR_INPUT
END_VAR
MotionCoupleTaskGearing.GearIn := FALSE;
MotionCoupleTaskGearing.Execute();
END_METHOD

{attribute 'monitoring' := 'call'}
PROPERTY GearRatioMaster1 : LREAL
SET
MotionCoupleTaskGearing.GearRatioMaster1 := GearRatioMaster1;
END_SET
END_PROPERTY

{attribute 'monitoring' := 'call'}
PROPERTY GearRatioMaster2 : LREAL
SET
MotionCoupleTaskGearing.GearRatioMaster2 := GearRatioMaster2;
END_SET
END_PROPERTY

{attribute 'monitoring' := 'call'}
PROPERTY GearRatioMaster3 : LREAL
SET
MotionCoupleTaskGearing.GearRatioMaster3 := GearRatioMaster3;
END_SET
END_PROPERTY

{attribute 'monitoring' := 'call'}
PROPERTY GearRatioMaster4 : LREAL
SET
MotionCoupleTaskGearing.GearRatioMaster4 := GearRatioMaster4;
END_SET
END_PROPERTY

PROPERTY Master1 : I_Axis
SET
MotionCoupleTaskGearing.Master1 := Master1;
END_SET
END_PROPERTY

PROPERTY Master2 : I_Axis
SET
MotionCoupleTaskGearing.Master2 := Master2;
END_SET
END_PROPERTY

PROPERTY Master3 : I_Axis
SET
MotionCoupleTaskGearing.Master3 := Master3;
END_SET
END_PROPERTY

PROPERTY Master4 : I_Axis
SET
MotionCoupleTaskGearing.Master4 := Master4;
END_SET
END_PROPERTY

END_FUNCTION_BLOCK

// Project Information/F_GetCompany
// This function has been automatically generated from the project information.
{attribute 'signature_flag' := '1073741824'}
{attribute 'TcGenerated'}
{attribute 'no-analysis'}
FUNCTION F_GetCompany : WSTRING
VAR_INPUT
	
END_VAR

F_GetCompany := "Beckhoff Automation LLC";

END_FUNCTION

// Project Information/F_GetTitle
// This function has been automatically generated from the project information.
{attribute 'signature_flag' := '1073741824'}
{attribute 'TcGenerated'}
{attribute 'no-analysis'}
FUNCTION F_GetTitle : WSTRING
VAR_INPUT
	
END_VAR

F_GetTitle := "ApplicationBase";

END_FUNCTION

// Project Information/F_GetVersion
// This function has been automatically generated from the project information.
{attribute 'signature_flag' := '1073741824'}
{attribute 'TcGenerated'}
{attribute 'no-analysis'}
FUNCTION F_GetVersion : ST_LibVersion
VAR_INPUT
	
END_VAR

F_GetVersion.iMajor := 1;
F_GetVersion.iMinor := 0;
F_GetVersion.iBuild := 8;
F_GetVersion.iRevision := 0;
F_GetVersion.sVersion := '1.0.8';
F_GetVersion.nFlags := 0;

END_FUNCTION

// Statemachine/Generic/SetStep
FUNCTION SetStep : UDINT
VAR_IN_OUT
	StateVar : UDINT;
END_VAR

VAR_INPUT
	Step : UDINT;
END_VAR

SetStep := StateVar := Step;

END_FUNCTION

// Statemachine/Generic/Statemachine_HMI
FUNCTION_BLOCK Statemachine_HMI EXTENDS HmiFunction
VAR
	Statemachine : I_Statemachine;
	{ attribute 'TcHmiSymbol.AddSymbol' }
	{ attribute 'TcHmiSymbol.AddSymbol.UserGroups' := '__SystemAdministrators,Admin' }
	Statemachine_HMI : ST_Statemachine_HMI;
END_VAR

PROPERTY ControlObject : I_Base
SET
__QueryInterface(ControlObject,Statemachine);
END_SET
END_PROPERTY

METHOD CyclicLogic
VAR_INST
	LastModeChangeCommand  : DINT;
	LastStateChangeCommand : DINT;
END_VAR
Statemachine_HMI.Name		  := Statemachine.Name;
Statemachine_HMI.CurrentState := Statemachine.CurrentState;
Statemachine_HMI.CurrentMode  := Statemachine.Mode.CurrentMode;
Statemachine_HMI.HmiEnabled	  := Enabled;
IF Enabled THEN
	IF Statemachine_HMI.ModeChangeCommand <> 0 THEN
		Statemachine.Mode.ChangeMode(Statemachine_HMI.ModeChangeCommand);
		LastModeChangeCommand			   := Statemachine_HMI.ModeChangeCommand;
		Statemachine_HMI.ModeChangeCommand := 0;
	END_IF

	{warning disable C0196}
	IF Statemachine_HMI.StateChangeCommand <> 0 THEN
		Statemachine.ChangeState(TO_UDINT(Statemachine_HMI.StateChangeCommand));
		{warning disable C0195}
		LastStateChangeCommand				:= Statemachine_HMI.StateChangeCommand;
		Statemachine_HMI.StateChangeCommand := 0;
	END_IF
ELSE
	Statemachine_HMI.StateChangeCommand := 0;
	Statemachine_HMI.ModeChangeCommand	:= 0;
END_IF
END_METHOD

(*FB_Init is always available implicitly and it is used primarily for initialization.
The return value is not evaluated. For a specific influence, you can also declare the
methods explicitly and provide additional code there with the standard initialization
code. You can evaluate the return value.*)
METHOD FB_Init : BOOL
VAR_INPUT
	(* TRUE: the retain variables are initialized (reset warm / reset cold)*)
	bInitRetains : BOOL;

	(* TRUE: the instance will be copied to the copy code afterward (online change)   *)
	bInCopyCode	 : BOOL;
	Name		 : T_MaxString;
	Statemachine : I_Statemachine;
END_VAR
THIS^.Statemachine := Statemachine;
ControlType		   := 'Statemachine';
LinkObject		   := 'Statemachine_HMI';
END_METHOD

END_FUNCTION_BLOCK

// Statemachine/PackML/NextAvailablePackMLCommands
FUNCTION_BLOCK NextAvailablePackMLCommands
VAR
	NextAvailableCommands : ARRAY[0..MAX_AVAILABLE_COMMANDS] OF E_PMLCommand;
	i					  : UDINT;
END_VAR

VAR CONSTANT
	MAX_AVAILABLE_COMMANDS : UDINT := 9;
END_VAR

METHOD PUBLIC GetCommands : ARRAY[0..MAX_AVAILABLE_COMMANDS] OF E_PMLCommand
VAR_INPUT
	CurrentMode	 : DINT(0..31);
	CurrentState : E_PMLState;
END_VAR

VAR
	ModeConfiguration : Tc3_PackML_V3.ST_PMLUnitModeConfiguration;
END_VAR
FOR i := 1 TO MAX_AVAILABLE_COMMANDS DO
	NextAvailableCommands[i] := E_PMLCommand.Undefined;
END_FOR

i				  := 0;
ModeConfiguration := Tc3_PackML_V3.GlobalVariables.stPMLUnitModeConfiguration[CurrentMode];
// Generate next possible Commands
CASE CurrentState OF
	E_PMLState.Undefined:
		;

	E_PMLState.Aborting:
		;

	E_PMLState.Aborted:
		NextAvailableCommands[i] := E_PMLCommand.Clear;

	E_PMLState.Clearing:
		;

	E_PMLState.Stopping:
		NextAvailableCommands[i] := E_PMLCommand.Abort;

	E_PMLState.Stopped:
		NextAvailableCommands[i] := E_PMLCommand.Abort;
		i						 := i + 1;
		IF NOT ModeConfiguration.aStateDisabled[E_PMLState.Resetting] AND NOT ModeConfiguration.aStateDisabled[E_PMLState.Idle] THEN
			NextAvailableCommands[i] := E_PMLCommand.Reset;
		ELSE
			NextAvailableCommands[i] := E_PMLCommand.Start;
		END_IF

	E_PMLState.Resetting:
		NextAvailableCommands[i] := E_PMLCommand.Abort;
		i						 := i + 1;
		NextAvailableCommands[i] := E_PMLCommand.Stop;

	E_PMLState.Idle:
		NextAvailableCommands[i] := E_PMLCommand.Abort;
		i						 := i + 1;
		NextAvailableCommands[i] := E_PMLCommand.Stop;
		i						 := i + 1;
		NextAvailableCommands[i] := E_PMLCommand.Start;

	E_PMLState.Starting:
		NextAvailableCommands[i] := E_PMLCommand.Abort;
		i						 := i + 1;
		NextAvailableCommands[i] := E_PMLCommand.Stop;

	E_PMLState.Execute:
		NextAvailableCommands[i] := E_PMLCommand.Abort;
		i						 := i + 1;
		NextAvailableCommands[i] := E_PMLCommand.Stop;
		i						 := i + 1;
		IF (NOT ModeConfiguration.aStateDisabled[E_PMLState.Held] AND NOT ModeConfiguration.aStateDisabled[E_PMLState.Holding]) OR (NOT ModeConfiguration.aStateDisabled[E_PMLState.Held] AND NOT ModeConfiguration.aStateDisabled[E_PMLState.Unholding]) THEN
			NextAvailableCommands[i] := E_PMLCommand.Hold;
			i						 := i + 1;
		END_IF

		IF (NOT ModeConfiguration.aStateDisabled[E_PMLState.Suspended] AND NOT ModeConfiguration.aStateDisabled[E_PMLState.Suspending]) OR (NOT ModeConfiguration.aStateDisabled[E_PMLState.Suspended] AND NOT ModeConfiguration.aStateDisabled[E_PMLState.Unsuspending]) THEN
			NextAvailableCommands[i] := E_PMLCommand.Suspend;
			i						 := i + 1;
		END_IF

		IF NOT ModeConfiguration.aStateDisabled[E_PMLState.Completed] AND NOT ModeConfiguration.aStateDisabled[E_PMLState.Completing] THEN
			NextAvailableCommands[i] := E_PMLCommand.Complete;
			i						 := i + 1;
		ELSIF NOT ModeConfiguration.aStateDisabled[E_PMLState.Resetting] THEN
			NextAvailableCommands[i] := E_PMLCommand.Reset;
			i						 := i + 1;
		END_IF

	E_PMLState.Completing:
		NextAvailableCommands[i] := E_PMLCommand.Abort;
		i						 := i + 1;
		NextAvailableCommands[i] := E_PMLCommand.Stop;

	E_PMLState.Completed:
		NextAvailableCommands[i] := E_PMLCommand.Abort;
		i						 := i + 1;
		NextAvailableCommands[i] := E_PMLCommand.Stop;
		i						 := i + 1;
		IF NOT ModeConfiguration.aStateDisabled[E_PMLState.Resetting] AND NOT ModeConfiguration.aStateDisabled[E_PMLState.Idle] THEN
			NextAvailableCommands[i] := E_PMLCommand.Reset;
		ELSE
			NextAvailableCommands[i] := E_PMLCommand.Start;
		END_IF

	E_PMLState.Holding:
		NextAvailableCommands[i] := E_PMLCommand.Abort;
		i						 := i + 1;
		NextAvailableCommands[i] := E_PMLCommand.Stop;

	E_PMLState.Held:
		NextAvailableCommands[i] := E_PMLCommand.Abort;
		i						 := i + 1;
		NextAvailableCommands[i] := E_PMLCommand.Stop;
		i						 := i + 1;
		NextAvailableCommands[i] := E_PMLCommand.Unhold;

	E_PMLState.Unholding:
		NextAvailableCommands[i] := E_PMLCommand.Abort;
		i						 := i + 1;
		NextAvailableCommands[i] := E_PMLCommand.Stop;

	E_PMLState.Suspending:
		NextAvailableCommands[i] := E_PMLCommand.Abort;
		i						 := i + 1;
		NextAvailableCommands[i] := E_PMLCommand.Stop;

	E_PMLState.Suspended:
		NextAvailableCommands[i] := E_PMLCommand.Abort;
		i						 := i + 1;
		NextAvailableCommands[i] := E_PMLCommand.Stop;
		i						 := i + 1;
		NextAvailableCommands[i] := E_PMLCommand.Unsuspend;

	E_PMLState.Unsuspending:
		NextAvailableCommands[i] := E_PMLCommand.Abort;
		i						 := i + 1;
		NextAvailableCommands[i] := E_PMLCommand.Stop;
END_CASE

GetCommands := NextAvailableCommands;
END_METHOD

END_FUNCTION_BLOCK

// Statemachine/PackML/PackMLStatemachine
FUNCTION_BLOCK PackMLStatemachine EXTENDS CyclicComponent IMPLEMENTS I_StateMachine
VAR
	StateList	   : StateList<17>;
	StateMachine   : FB_PMLStateMachine;
	StateCommand   : E_PMLCommand;
	_CurrentState  : E_PMLState;
	ModeController : PackMLModeControl := (StateMachine := THIS^);
END_VAR

PROPERTY Mode : I_Mode
GET
Mode := ModeController;
END_GET
SET
// Fix defined in PackML
END_SET
END_PROPERTY

METHOD PROTECTED CallState : BOOL
VAR_INPUT
	StateIndex : E_PMLState;
END_VAR

VAR
	State : I_State;
	i	  : DINT;
END_VAR
State := StateList.GetStateAtIndex(StateIndex);
IF State <> 0 THEN
	CallState := State.Executing();
ELSE
	CallState := TRUE;
END_IF

FOR i := 0 TO StateList.NumberOfStates DO
	State := StateList.GetStateAtIndex(i);
	IF State <> 0 AND i <> StateIndex THEN
		State.Inactive();
	END_IF
END_FOR
END_METHOD

METHOD ChangeState
VAR_INPUT
	StateCommand : DINT;
END_VAR
IF StateCommand <= 0 OR StateCommand > 17 THEN
	Trace.LogMessage('PackML Statemachine ChangeState()', 'StateId is not a PackML State');
END_IF

{warning disable C0196}
THIS^.StateCommand := StateCommand;
END_METHOD

{attribute 'monitoring' := 'call'}
PROPERTY CurrentState : DINT
GET
CurrentState := _CurrentState;
END_GET
END_PROPERTY

PROPERTY States : I_StateList
GET
States := StateList;
END_GET
END_PROPERTY

METHOD CyclicLogic
VAR_INST
	ClearingTon : TON;
END_VAR
IF StateList.NumberOfStates = 0 THEN
	RETURN;
END_IF

ModeController.CyclicLogic();
IF _CurrentState = E_PMLState.Undefined AND Mode.CurrentMode <> 0 THEN
	StateCommand := E_PMLCommand.Abort;
END_IF

StateMachine(eMode			  := TO_DINT(Mode.CurrentMode),
			 eCommand		  := StateCommand,
			 stSubUnitInfoRef :=,
			 stOptions		  :=,
			 eState			  => _CurrentState,
			 sState			  =>,
			 bError			  =>,
			 nErrorID		  =>);

CASE _CurrentState OF
	E_PMLState.Undefined:
		CallState(_CurrentState);

	E_PMLState.Clearing:
		ClearingTon(IN := TRUE, PT := ApplicationBaseParameter.ClearingTimeout);
		IF CallState(_CurrentState) THEN
			ClearingTon(IN := FALSE);
			StateMachine.M_StateComplete();
		END_IF

		IF ClearingTon.Q THEN
			ClearingTon(IN := FALSE);
			Trace.LogMessage('Clearing Timeout exeeded!', 'ApplicationBaseParameter.ClearingTimeout');
			StateCommand := E_PMLCommand.Abort;
		END_IF

	E_PMLState.Stopped:
		CallState(_CurrentState);

	E_PMLState.Starting:
		IF CallState(_CurrentState) THEN
			StateMachine.M_StateComplete();
		END_IF

	E_PMLState.Idle:
		CallState(_CurrentState);

	E_PMLState.Suspended:
		CallState(_CurrentState);

	E_PMLState.Execute:
		CallState(_CurrentState);

	E_PMLState.Stopping:
		IF CallState(_CurrentState) THEN
			StateMachine.M_StateComplete();
		END_IF

	E_PMLState.Aborting:
		IF CallState(_CurrentState) THEN
			StateMachine.M_StateComplete();
		END_IF

	E_PMLState.Aborted:
		CallState(_CurrentState);

	E_PMLState.Holding:
		IF CallState(_CurrentState) THEN
			StateMachine.M_StateComplete();
		END_IF

	E_PMLState.Held:
		CallState(_CurrentState);

	E_PMLState.Unholding:
		IF CallState(_CurrentState) THEN
			StateMachine.M_StateComplete();
		END_IF

	E_PMLState.Suspending:
		IF CallState(_CurrentState) THEN
			StateMachine.M_StateComplete();
		END_IF

	E_PMLState.Unsuspending:
		IF CallState(_CurrentState) THEN
			StateMachine.M_StateComplete();
		END_IF

	E_PMLState.Resetting:
		IF CallState(_CurrentState) THEN
			StateMachine.M_StateComplete();
		END_IF

	E_PMLState.Completing:
		IF CallState(_CurrentState) THEN
			StateMachine.M_StateComplete();
		END_IF

	E_PMLState.Completed:
		CallState(_CurrentState);
END_CASE
END_METHOD

END_FUNCTION_BLOCK

// Statemachine/PackML/PackMLStatemachine_HMI
FUNCTION_BLOCK PackMLStatemachine_HMI EXTENDS HmiFunction
VAR
	Statemachine				: I_Statemachine;
	NextAvailablePackMLCommands : NextAvailablePackMLCommands;
	{ attribute 'TcHmiSymbol.AddSymbol' }
	{ attribute 'TcHmiSymbol.AddSymbol.UserGroups' := '__SystemAdministrators,Admin' }
	Statemachine_HMI : ST_PackMLStatemachine_HMI;
END_VAR

PROPERTY ControlObject : I_Base
SET
__QueryInterface(ControlObject,Statemachine);
END_SET
END_PROPERTY

METHOD CyclicLogic
VAR_INST
	LastModeChangeCommand  : DINT;
	LastStateChangeCommand : UDINT;
END_VAR
{warning disable C0196}
Statemachine_HMI.CurrentState := Statemachine.CurrentState;
Statemachine_HMI.CurrentMode  := Statemachine.Mode.CurrentMode;
Statemachine_HMI.Name		  := Statemachine.Name;
Statemachine_HMI.HmiEnabled	  := Enabled;
IF Enabled THEN
	IF Statemachine_HMI.ModeCommand <> 0 THEN
		Statemachine.Mode.ChangeMode(Statemachine_HMI.ModeCommand);
		LastModeChangeCommand		 := Statemachine_HMI.ModeCommand;
		Statemachine_HMI.ModeCommand := 0;
	END_IF

	{warning disable C0196}
	IF Statemachine_HMI.StateCommand <> 0 THEN
		Statemachine.ChangeState(TO_UDINT(Statemachine_HMI.StateCommand));
		{warning disable C0195}
		LastStateChangeCommand		  := Statemachine_HMI.StateCommand;
		Statemachine_HMI.StateCommand := 0;
	END_IF
ELSE
	Statemachine_HMI.StateCommand := 0;
	Statemachine_HMI.ModeCommand  := 0;
END_IF

Statemachine_HMI.NextAvailableCommands := NextAvailablePackMLCommands.GetCommands(Statemachine_HMI.CurrentMode, Statemachine_HMI.CurrentState);
END_METHOD

(*FB_Init is always available implicitly and it is used primarily for initialization.
The return value is not evaluated. For a specific influence, you can also declare the
methods explicitly and provide additional code there with the standard initialization
code. You can evaluate the return value.*)
METHOD FB_Init : BOOL
VAR_INPUT
	(* TRUE: the retain variables are initialized (reset warm / reset cold)*)
	bInitRetains : BOOL;

	(* TRUE: the instance will be copied to the copy code afterward (online change)   *)
	bInCopyCode	 : BOOL;
	Name		 : T_MaxString;
	Statemachine : I_Statemachine;
END_VAR
THIS^.Statemachine := Statemachine;
ControlType		   := 'PackMLStatemachine';
LinkObject		   := 'Statemachine_HMI';
END_METHOD

END_FUNCTION_BLOCK

// Utilities/AnyBuffer/Interface/I_AnyBuffer
INTERFACE I_AnyBuffer

// Clears all buffer data and resets metadata to initial state
METHOD Clear : BOOL
END_METHOD

PROPERTY Configuration : REFERENCE TO ST_BufferConfiguration
GET
END_GET
END_PROPERTY

// Deletes element at specified index position and decrements element count
METHOD DeleteAtIndex : BOOL
VAR_INPUT
	index : DINT; // Zero-based index position of element to delete
END_VAR
END_METHOD

PROPERTY isEmpty : BOOL
GET
END_GET
END_PROPERTY

PROPERTY isFull : BOOL
GET
END_GET
END_PROPERTY

PROPERTY Metadata : REFERENCE TO ST_BufferMetadata
GET
END_GET
END_PROPERTY

// Retrieve an element at a specific index without removing it from the buffer
METHOD PeekAtIndex : BOOL
VAR_INPUT
	index	: DINT;
	element : ANY;
END_VAR
END_METHOD

// Remove and retrieve an element at a specific index, shifting remaining elements left
METHOD PopAtIndex : BOOL
VAR_INPUT
	index	   : DINT;
	element	   : ANY;
	popDiscard : BOOL := FALSE;
END_VAR
END_METHOD

// Removes and retrieves the first element from the buffer (FIFO/queue operation)
METHOD PopLeft : BOOL
VAR_INPUT
	element	   : ANY;			// Variable to receive the popped element
	popDiscard : BOOL := FALSE; // When TRUE, element is removed but not copied (type checking skipped)
END_VAR
END_METHOD

// Removes and retrieves the last element from the buffer (stack pop operation)
METHOD PopRight : BOOL
VAR_INPUT
	element	   : ANY;			// Variable to receive the popped element
	popDiscard : BOOL := FALSE; // When TRUE, element is removed but not copied (type checking skipped)
END_VAR
END_METHOD

// Add an element at a specific index, shifting remaining elements right
METHOD PushAtIndex : BOOL
VAR_INPUT
	index	: DINT;
	element : ANY;
END_VAR
END_METHOD

// Appends a new element to the left side of the buffer (LIFO/stack push operation)
METHOD PushLeft : BOOL
VAR_INPUT
	element : ANY;
END_VAR
END_METHOD

// Appends a new element to the right side of the buffer (FIFO/queue enqueue operation)
METHOD PushRight : BOOL
VAR_INPUT
	element : ANY;
END_VAR
END_METHOD

// Replaces an element at a specific index with the given element
METHOD ReplaceAtIndex : BOOL
VAR_INPUT
	index	: DINT;
	element : ANY;
END_VAR
END_METHOD

END_INTERFACE

// Utilities/AnyBuffer/Interface/I_AnyBufferStrategy
INTERFACE I_AnyBufferStrategy

METHOD Clear : BOOL
END_METHOD

PROPERTY isEmpty : BOOL
GET
END_GET
END_PROPERTY

PROPERTY isFull : BOOL
GET
END_GET
END_PROPERTY

END_INTERFACE

// Utilities/AnyBuffer/TypedBuffers/FifoBuffer
// Provides a simplified FIFO queue interface as an adapter over AnyBuffer
FUNCTION_BLOCK FifoBuffer IMPLEMENTS I_AnyBufferStrategy
VAR
	anyBuffer	  : I_AnyBuffer;
	isInitialized : BOOL := FALSE;
	_overwrite	  : BOOL := FALSE; // When TRUE, Push overwrites oldest element when full
	_reversed	  : BOOL := FALSE; // When TRUE, reverses push/pop direction (PushLeft/PopRight)
	{attribute 'hide'}
	discardObject : BYTE; // element for discarding elements in overwrite mode
END_VAR

(*
## Detailed Description

FifoBuffer is an adapter (also known as a strategy or facade) that wraps an AnyBuffer instance
to provide a simplified First-In-First-Out (FIFO) queue interface. Instead of using the full
AnyBuffer API with directional operations (AppendLeft/Right, PopLeft/Right), users can simply
Push and Pop elements following standard queue semantics.

### Alternative Names
In computer science, FIFO data structures are commonly called "Queues". This implementation
could alternatively be named "Queue" or "QueueAdapter" for more conventional naming.

### Design Pattern
This implements the **Adapter Pattern** (also Strategy Pattern), which:
- Wraps a more complex interface (I_AnyBuffer) with a simpler, domain-specific interface
- Delegates all operations to the underlying AnyBuffer instance
- Provides semantic clarity: Push/Pop vs AppendLeft/PopRight
- Allows multiple strategy implementations (FIFO, LIFO, Priority, etc.) over the same buffer

### FIFO Semantics
- **Push(element)**: Adds element using PushRight (reversed=FALSE) or PushLeft (reversed=TRUE)
- **Pop(element)**: Removes element using PopLeft (reversed=FALSE) or PopRight (reversed=TRUE)
- The reversed parameter controls the direction of both Push and Pop operations
- Elements maintain insertion order, but retrieval order depends on reversed setting

### Configurable Behavior
The FifoBuffer supports two optional parameters during initialization:

**overwrite parameter:**
- **FALSE (default)**: Push fails when buffer is full, returns FALSE and logs error
- **TRUE**: Push to full buffer automatically removes element to make space (circular buffer behavior)
  - When reversed=FALSE: Removes from front (PopLeft), adds to back (PushRight)
  - When reversed=TRUE: Removes from back (PopRight), adds to front (PushLeft)
  - Removed element is discarded using internal temporary buffer

**reversed parameter:**
- **FALSE (default)**: Standard FIFO - Push to back (PushRight), Pop from front (PopLeft)
- **TRUE**: Reversed direction - Push to front (PushLeft), Pop from back (PopRight)
- When reversed=TRUE, behavior is similar to LIFO/stack but with directional consistency

### Operation Mapping
**Standard Mode (overwrite=FALSE, reversed=FALSE):**
```
Push()  -> anyBuffer.PushRight()  // Add to back (right)
Pop()   -> anyBuffer.PopLeft()    // Remove from front (left)
Clear() -> anyBuffer.Clear()      // Clear all
isEmpty -> anyBuffer.isEmpty      // Check if empty
isFull  -> anyBuffer.isFull       // Check if full
```

**Overwrite Mode (overwrite=TRUE, reversed=FALSE):**
```
Push()  -> if full: anyBuffer.PopLeft(pBufferTemp), then anyBuffer.PushRight()
Pop()   -> anyBuffer.PopLeft()    // Remove from front (left)
```

**Reversed Mode (overwrite=FALSE, reversed=TRUE):**
```
Push()  -> anyBuffer.PushLeft()   // Add to front (left)
Pop()   -> anyBuffer.PopRight()   // Remove from back (right)
```

**Overwrite + Reversed Mode (overwrite=TRUE, reversed=TRUE):**
```
Push()  -> if full: anyBuffer.PopRight(pBufferTemp), then anyBuffer.PushLeft()
Pop()   -> anyBuffer.PopRight()   // Remove from back (right)
```

### Usage Examples

**Standard FIFO Mode:**
```iecst
VAR
    rawBuffer : ARRAY[0..2] OF DINT;
    buffer : AnyBuffer(pBuffer := rawBuffer,
                       bufferBoundLower := 0,
                       bufferBoundUpper := 2,
                       isBufferPersistent := FALSE);
    fifo : FifoBuffer(anyBuffer := buffer, overwrite := FALSE, reversed := FALSE);
    value : DINT;
END_VAR

// Push elements
value := 100; fifo.Push(value);  // Queue: [100]
value := 200; fifo.Push(value);  // Queue: [100, 200]
value := 300; fifo.Push(value);  // Queue: [100, 200, 300]

// Pop elements (FIFO order - oldest first)
fifo.Pop(value);   // value = 100, Queue: [200, 300]
fifo.Pop(value);   // value = 200, Queue: [300]
fifo.Pop(value);   // value = 300, Queue: []
```

**Overwrite Mode (Circular Buffer):**
```iecst
VAR
    fifo : FifoBuffer(anyBuffer := buffer, overwrite := TRUE, reversed := FALSE);
END_VAR

// Fill buffer
value := 100; fifo.Push(value);  // Queue: [100]
value := 200; fifo.Push(value);  // Queue: [100, 200]
value := 300; fifo.Push(value);  // Queue: [100, 200, 300]

// Push to full buffer overwrites oldest
value := 400; fifo.Push(value);  // Queue: [200, 300, 400] - 100 was removed
value := 500; fifo.Push(value);  // Queue: [300, 400, 500] - 200 was removed
```

**Reversed Mode (reversed=TRUE):**
```iecst
VAR
    fifo : FifoBuffer(anyBuffer := buffer, overwrite := FALSE, reversed := TRUE);
END_VAR

// Push elements (adds to front using PushLeft)
value := 100; fifo.Push(value);  // Buffer: [100]
value := 200; fifo.Push(value);  // Buffer: [200, 100] - 200 added to front
value := 300; fifo.Push(value);  // Buffer: [300, 200, 100] - 300 added to front

// Pop elements (removes from back using PopRight)
fifo.Pop(value);   // value = 100, Buffer: [300, 200]
fifo.Pop(value);   // value = 200, Buffer: [300]
fifo.Pop(value);   // value = 300, Buffer: []
```

### Advantages
- **Simplified interface**: Push/Pop instead of AppendLeft/PopRight
- **Semantic clarity**: Code intention is clearer with queue terminology
- **Flexibility**: Easy to swap different buffer strategies (FIFO, LIFO, etc.)
- **Type safety**: Enforces FIFO semantics at compile time through interface

### Limitations
- No random access: Cannot peek at arbitrary indices (use AnyBuffer directly if needed)
- No priority queue: Elements are strictly ordered by insertion time
- Overwrite mode loses oldest data when buffer is full
- Combining overwrite and reversed modes creates a circular stack behavior

### Dependencies
- Requires I_AnyBuffer implementation (e.g., AnyBuffer)
- Uses Trace for error logging and verbose diagnostics
- Implements I_AnyBufferStrategy interface

### Related Patterns
- **LifoBuffer**: Would implement stack (Last-In-First-Out) semantics
- **PriorityBuffer**: Would implement priority queue with ordered insertion
- **CircularBuffer**: Would implement ring buffer with overwrite semantics
*)

// Removes all elements from the queue and resets to empty state
METHOD Clear : BOOL

(*
## Detailed Description

Clears all elements from the underlying buffer, resetting it to an empty state.
After calling Clear, isEmpty will return TRUE and elementCount will be 0.

This operation delegates directly to the underlying anyBuffer.Clear() method.

### Return Value
- **TRUE**: Queue was successfully cleared
- **FALSE**: Clear operation failed (e.g., anyBuffer is not initialized)

### Side Effects
- All elements are removed from the buffer
- Element count is reset to 0
- Buffer capacity is restored to maximum
- Logs verbose trace message on success
*)
Clear := FALSE;
IF anyBuffer <> 0 THEN
	Clear := anyBuffer.Clear();
	;
END_IF

Trace.Verbose(__POUNAME(), 'executed');
END_METHOD

// Initializes the FIFO queue by injecting the underlying buffer dependency
METHOD FB_Init : BOOL
VAR_INPUT
	bInitRetains : BOOL;		// TRUE: the retain variables are initialized (reset warm / reset cold)
	bInCopyCode	 : BOOL;		// TRUE: the instance will be copied to the copy code afterward (online change)
	anyBuffer	 : I_AnyBuffer; // The underlying buffer implementation to wrap
	overwrite	 : BOOL;		// When TRUE, Push overwrites oldest element when full
	reversed	 : BOOL;		// When TRUE, reverses push/pop direction (PushLeft/PopRight)
END_VAR

(*
## Detailed Description

Initializes the FifoBuffer by injecting the underlying AnyBuffer dependency. This follows
the dependency injection pattern where the buffer implementation is provided during
construction rather than being created internally.

### Initialization Sequence
1. Validates that a valid anyBuffer reference is provided (non-zero pointer)
2. Stores the buffer reference for use by Push, Pop, and other operations
3. Sets isInitialized flag to TRUE to enable operations

### Parameters
- **anyBuffer**: Reference to an I_AnyBuffer implementation (e.g., AnyBuffer instance)
  - Must be a valid, initialized buffer
  - This FifoBuffer will delegate all operations to this buffer
- **overwrite**: Controls behavior when pushing to a full buffer
  - **FALSE (default)**: Push returns FALSE and logs error when buffer is full
  - **TRUE**: Push automatically removes an element to make space (circular buffer behavior)
    - When reversed=FALSE: Removes from front (PopLeft), adds to back (PushRight)
    - When reversed=TRUE: Removes from back (PopRight), adds to front (PushLeft)
  - Discarded element is popped to internal temporary buffer (pBufferTemp)
- **reversed**: Controls the direction of both Push and Pop operations
  - **FALSE (default)**: Push to back (PushRight), Pop from front (PopLeft) - standard FIFO
  - **TRUE**: Push to front (PushLeft), Pop from back (PopRight) - reversed direction
  - Affects the operational direction of the buffer, not just retrieval order

### Return Value
Returns BOOL but value is not evaluated by the runtime. Always call with valid anyBuffer.

### Usage Example
```iecst
VAR
    rawBuffer : ARRAY[0..9] OF DINT;
    buffer : AnyBuffer(pBuffer := rawBuffer,
                       bufferBoundLower := 0,
                       bufferBoundUpper := 9,
                       isBufferPersistent := FALSE);
    fifo : FifoBuffer(anyBuffer := buffer,
                      overwrite := FALSE,
                      reversed := FALSE);
END_VAR
```

### Important Notes
- Must provide a valid anyBuffer reference, otherwise Push/Pop will fail
- The underlying buffer must already be initialized before passing to FB_Init
- A temporary buffer (pBufferTemp) is allocated internally for discarding elements in overwrite mode
- pBufferTemp is automatically deallocated in FB_exit
- Overwrite mode is useful for logging/telemetry where newest data is more important
- Reversed mode changes the operational direction of both Push and Pop
- Combining overwrite=TRUE and reversed=TRUE creates a circular buffer operating from the opposite end
*)
IF anyBuffer <> 0 THEN
	THIS^.anyBuffer := anyBuffer;
	_overwrite		:= overwrite;
	_reversed		:= reversed;
	isInitialized	:= TRUE;
END_IF
END_METHOD

// Returns TRUE if the queue contains no elements
PROPERTY isEmpty : BOOL

(*
## Detailed Description

Returns TRUE if the queue is empty (contains no elements), FALSE otherwise.
This property delegates directly to the underlying anyBuffer.isEmpty property.

Use this property to check if Pop operation would succeed before attempting to
remove an element.

### Return Value
- **TRUE**: Queue is empty (elementCount = 0)
- **FALSE**: Queue contains one or more elements

### Usage Example
```iecst
IF NOT fifo.isEmpty THEN
    fifo.Pop(value);  // Safe to pop
END_IF
```
*)
GET
isEmpty := anyBuffer.isEmpty;
END_GET
END_PROPERTY

// Returns TRUE if the queue is at maximum capacity
PROPERTY isFull : BOOL

(*
## Detailed Description

Returns TRUE if the queue is full (at maximum capacity), FALSE otherwise.
This property delegates directly to the underlying anyBuffer.isFull property.

Use this property to check if Push operation would succeed before attempting to
add an element.

### Return Value
- **TRUE**: Queue is full (elementCount = capacity)
- **FALSE**: Queue has space for more elements

### Usage Example
```iecst
IF NOT fifo.isFull THEN
    value := 100;
    fifo.Push(value);  // Safe to push
END_IF
```
*)
GET
isFull := anyBuffer.isFull;
END_GET
END_PROPERTY

// Removes and retrieves an element from the queue (FIFO or LIFO depending on reversed setting)
{attribute 'hasanytype'}
METHOD Pop : BOOL
VAR_INPUT
	element : ANY; // Variable to receive the popped element
END_VAR

(*
## Detailed Description

Removes and retrieves an element from the queue. The behavior depends on the 'reversed'
initialization parameter:

**When reversed = FALSE (default mode):**
- Removes element from the front (left side, index 0)
- Delegates to anyBuffer.PopLeft()
- Standard FIFO behavior when combined with PushRight

**When reversed = TRUE (reversed mode):**
- Removes element from the back (right side, highest index)
- Delegates to anyBuffer.PopRight()
- Reversed direction - removes from opposite end compared to default
- Combined with PushLeft, maintains FIFO order but from opposite direction

### Operation Sequence
1. Validates that the buffer has been initialized
2. Validates that element size matches the buffer's configured element size
3. Checks that the queue is not empty
4. Removes element using PopLeft (FIFO) or PopRight (LIFO) based on reversed setting
5. Copies the element value to the output parameter
6. For PopLeft: Shifts remaining elements left; For PopRight: No shifting needed
7. Logs verbose trace on success or error trace on failure

### Standard Mode Example (reversed = FALSE)
```iecst
// Push to right, Pop from left
value := 100; fifo.Push(value);  // Buffer: [100]
value := 200; fifo.Push(value);  // Buffer: [100, 200] - 200 added to right
value := 300; fifo.Push(value);  // Buffer: [100, 200, 300] - 300 added to right

fifo.Pop(value);  // Returns 100 (from left), Buffer: [200, 300]
fifo.Pop(value);  // Returns 200 (from left), Buffer: [300]
fifo.Pop(value);  // Returns 300 (from left), Buffer: []
```

### Reversed Mode Example (reversed = TRUE)
```iecst
// Push to left, Pop from right
value := 100; fifo.Push(value);  // Buffer: [100]
value := 200; fifo.Push(value);  // Buffer: [200, 100] - 200 added to left
value := 300; fifo.Push(value);  // Buffer: [300, 200, 100] - 300 added to left

fifo.Pop(value);  // Returns 100 (from right), Buffer: [300, 200]
fifo.Pop(value);  // Returns 200 (from right), Buffer: [300]
fifo.Pop(value);  // Returns 300 (from right), Buffer: []
```

### Return Value
- **TRUE**: Element was successfully popped and copied to element parameter
- **FALSE**: Pop operation failed (see error conditions)

### Error Conditions
- Returns FALSE and logs error if buffer was not initialized
- Returns FALSE and logs error if element size doesn't match buffer element size
- Returns FALSE and logs error if queue is empty (no elements to pop)
- Returns FALSE and logs error if underlying PopLeft or PopRight operation fails

### Parameters
- **element**: Must be a writable variable (not a literal) of the correct size
  - Must match the buffer's configured element size
  - Will receive the popped element value on success

### Side Effects
- Removes one element from the queue
- Decrements element count by 1
- For FIFO mode (reversed=FALSE): Shifts remaining elements one position to the left
- For LIFO mode (reversed=TRUE): No element shifting required
- Logs verbose trace message on success
- Logs error trace message on failure
*)
Pop := FALSE;
IF NOT isInitialized THEN
	Trace.Error(__POUNAME(), 'Buffer was not initialized yet, execute method .init() at least once');
	RETURN;
END_IF

// valid sized element?
IF element.diSize <> anyBuffer.Configuration.elementSize THEN
	Trace.Error(__POUNAME(), 'Passed element to pop to is of improper size');
	RETURN;
END_IF

// retrieve element from buffer if there is any left
IF NOT isEmpty THEN
	IF _reversed THEN
		// LIFO mode: pop from back (newest first)
		Pop := anyBuffer.PopRight(element);
	ELSE
		// FIFO mode: pop from front (oldest first)
		Pop := anyBuffer.PopLeft(element);
	END_IF
ELSE
	Trace.Error(__POUNAME(), 'Attempt to pop from empty buffer');
END_IF

// Pop was ok, trace message
IF Pop THEN
	Trace.Verbose(__POUNAME(), 'executed');
ELSE
	Trace.Error(__POUNAME(), 'FAILED');
END_IF
END_METHOD

// Adds a new element to the queue (direction depends on reversed setting)
{attribute 'hasanytype'}
METHOD Push : BOOL
VAR_INPUT
	element : ANY; // Element to add to the queue
END_VAR

(*
## Detailed Description

Adds a new element to the queue. The push direction and overwrite behavior depend on
the 'reversed' and 'overwrite' initialization parameters.

**Push Direction (reversed parameter):**
- **reversed = FALSE (default)**: Delegates to anyBuffer.PushRight() - adds to back/right
- **reversed = TRUE**: Delegates to anyBuffer.PushLeft() - adds to front/left

**Overwrite Behavior (overwrite parameter):**
- **overwrite = FALSE (default)**: Push fails if buffer is full, returns FALSE and logs error
- **overwrite = TRUE (circular buffer mode)**: Push succeeds even when buffer is full
  - When reversed=FALSE: Removes element from front (PopLeft to pBufferTemp), then adds to back (PushRight)
  - When reversed=TRUE: Removes element from back (PopRight to pBufferTemp), then adds to front (PushLeft)
  - Discarded element is popped to internal temporary buffer and dropped
  - Useful for logging/telemetry where newest data is more important

### Operation Sequence

**Standard Mode (overwrite = FALSE, reversed = FALSE):**
1. Validates that the buffer has been initialized
2. Validates that element size matches the buffer's configured element size
3. Checks that the queue is not full (has available capacity)
4. If full: Returns FALSE and logs error
5. If not full: Adds element to the back using PushRight
6. Logs verbose trace on success or error trace on failure

**Standard Mode with Reversed (overwrite = FALSE, reversed = TRUE):**
1. Validates that the buffer has been initialized
2. Validates that element size matches the buffer's configured element size
3. Checks that the queue is not full (has available capacity)
4. If full: Returns FALSE and logs error
5. If not full: Adds element to the front using PushLeft
6. Logs verbose trace on success or error trace on failure

**Overwrite Mode (overwrite = TRUE, reversed = FALSE):**
1. Validates that the buffer has been initialized
2. Validates that element size matches the buffer's configured element size
3. If buffer is full: Removes oldest element using PopLeft (discards to pBufferTemp)
4. Adds new element to the back using PushRight
5. Logs verbose trace on success or error trace on failure

**Overwrite Mode with Reversed (overwrite = TRUE, reversed = TRUE):**
1. Validates that the buffer has been initialized
2. Validates that element size matches the buffer's configured element size
3. If buffer is full: Removes element using PopRight (discards to pBufferTemp)
4. Adds new element to the front using PushLeft
5. Logs verbose trace on success or error trace on failure

### Standard Mode Example (overwrite = FALSE)
```iecst
// Starting with empty queue
value := 100; fifo.Push(value);  // Queue: [100]
value := 200; fifo.Push(value);  // Queue: [100, 200]
value := 300; fifo.Push(value);  // Queue: [100, 200, 300]

// Pop operations retrieve in FIFO order (oldest first)
fifo.Pop(value);  // Returns 100 (first pushed)
fifo.Pop(value);  // Returns 200 (second pushed)
fifo.Pop(value);  // Returns 300 (third pushed)
```

### Overwrite Mode Example (overwrite = TRUE)
```iecst
// Assuming buffer capacity is 3
value := 100; fifo.Push(value);  // Queue: [100]
value := 200; fifo.Push(value);  // Queue: [100, 200]
value := 300; fifo.Push(value);  // Queue: [100, 200, 300] - full

// Push to full buffer overwrites oldest
value := 400; fifo.Push(value);  // Queue: [200, 300, 400] - 100 removed
value := 500; fifo.Push(value);  // Queue: [300, 400, 500] - 200 removed
```

### Return Value
- **TRUE**: Element was successfully pushed to the queue
- **FALSE**: Push operation failed (see error conditions)

### Error Conditions
- Returns FALSE and logs error if buffer was not initialized
- Returns FALSE and logs error if element size doesn't match buffer element size
- Returns FALSE and logs error if queue is full AND overwrite is FALSE
- Returns FALSE and logs error if underlying PushRight operation fails
- In overwrite mode, Push should always succeed unless buffer is not initialized or element size is wrong

### Parameters
- **element**: Must be a writable variable (not a literal) of the correct size
  - Must match the buffer's configured element size
  - Value will be copied into the queue

### Side Effects

**Standard Mode (overwrite = FALSE):**
- Adds one element to the queue at the back (next available index)
- No shifting of existing elements required
- Increments element count by 1
- Decrements available capacity by 1
- Logs verbose trace message on success
- Logs error trace message on failure

**Overwrite Mode (overwrite = TRUE):**
- If buffer is full: Removes oldest element first (PopLeft with shifting)
- Adds new element to the back (next available index)
- Element count remains constant when overwriting
- Logs verbose trace message on success
- Logs error trace message on failure

### Performance Considerations
- **Standard mode (reversed=FALSE)**: O(1) - PushRight is constant time, no shifting
- **Standard mode (reversed=TRUE)**: O(n) - PushLeft requires shifting all elements right
- **Overwrite mode (reversed=FALSE)**: O(n) when full (PopLeft + PushRight both with shifting)
- **Overwrite mode (reversed=TRUE)**: O(n) when full (PopRight O(1) + PushLeft O(n))
- **Overwrite mode**: O(1) or O(n) when not full (depends on reversed setting)
- Pop operation with reversed=FALSE has O(n) complexity (PopLeft with shifting)
- Pop operation with reversed=TRUE has O(1) complexity (PopRight, no shifting)
- Trade-off: reversed=FALSE optimizes Push, reversed=TRUE optimizes Pop
*)
Push := FALSE;
IF NOT isInitialized THEN
	Trace.Error(__POUNAME(), 'Buffer was not initialized yet, execute method .init() at least once');
	RETURN;
END_IF

// valid sized element pushed?
IF element.diSize <> anyBuffer.Configuration.elementSize THEN
	Trace.Error(__POUNAME(), 'Pushed element is of improper size');
	RETURN;
END_IF

// handle full buffer based on overwrite setting
IF isFull THEN
	IF _overwrite THEN
		// Overwrite mode: remove element to make space (discard to pBufferTemp)
		IF _reversed THEN
			// Reversed: remove from back before adding to front
			anyBuffer.PopRight(discardObject, TRUE);
		ELSE
			// Standard: remove from front before adding to back
			anyBuffer.PopLeft(discardObject, TRUE);
		END_IF
	ELSE
		// Standard mode: fail and log error
		Trace.Error(__POUNAME(), 'Attempt to push to full buffer');
		RETURN;
	END_IF
END_IF

// add element based on direction setting
IF _reversed THEN
	// Reversed: add to front (left)
	Push := anyBuffer.PushLeft(element);
ELSE
	// Standard: add to back (right)
	Push := anyBuffer.PushRight(element);
END_IF

// Push was ok, trace message
IF Push THEN
	Trace.Verbose(__POUNAME(), 'executed');
ELSE
	Trace.Error(__POUNAME(), 'FAILED');
END_IF
END_METHOD

END_FUNCTION_BLOCK

// Utilities/AnyBuffer/AnyBuffer
// the AnyBuffer block behaves as a double ended que

// elements can be appended / popped left and right
FUNCTION_BLOCK AnyBuffer IMPLEMENTS I_AnyBuffer
VAR
	bufferConfiguration : ST_BufferConfiguration;
	isInitialized		: BOOL := FALSE;
	pBuffer				: ANYTYPE;
	{attribute 'hide'}
	pBufferTemp : POINTER TO BYTE;
END_VAR

VAR PERSISTENT
	bufferMetadata : ST_BufferMetadata;
END_VAR

PROPERTY buffer : ANYTYPE
GET
buffer := pBuffer;
END_GET
END_PROPERTY

// Clears all buffer data and resets metadata to initial state
METHOD Clear : BOOL

(*
## Detailed Description

Clears all data from the buffer and resets the metadata to its initial state. This method
performs a complete buffer reset by zeroing out both the buffer contents and all tracking
metadata, effectively returning the buffer to an empty, initialized state.

### Operation Sequence
1. Validates that the buffer has been properly initialized via FB_init/Initialize
2. Clears all buffer data using memset (sets all bytes to 0x00)
3. Clears all metadata (elementCount, capacity, etc.) using memset
4. Logs success or failure via Trace system

### Key Features
- **Complete reset**: Zeros out both buffer data and metadata structures
- **Initialization check**: Validates buffer is initialized before attempting clear
- **Safe operation**: Cannot corrupt uninitialized or invalid buffers
- **Comprehensive logging**: Traces verbose success or error failure messages
- **Fast execution**: Uses memset for efficient memory clearing

### Usage Example
```iecst
VAR
    buffer : AnyBuffer(pBuffer := myArray, bufferBoundLower := 0, bufferBoundUpper := 9, isBufferPersistent := FALSE);
    success : BOOL;
END_VAR

// Add some data
buffer.PushRight(value1);
buffer.PushRight(value2);

// Clear all data
success := buffer.Clear();
IF success THEN
    // Buffer is now empty, elementCount = 0
    // All buffer positions are zeroed
END_IF
```

### Return Value
- **TRUE**: Buffer was successfully cleared (both data and metadata)
- **FALSE**: Clear operation failed (buffer not initialized)

### Error Conditions
- Returns FALSE and logs error if buffer was not properly initialized
- This prevents clearing invalid or uninitialized memory regions

### Side Effects
- Sets all buffer element positions to zero (0x00)
- Resets elementCount to 0
- Resets all other metadata fields to 0
- Buffer can be immediately reused after successful clear

### Dependencies
- Requires buffer to be initialized via FB_init or Initialize method
- Uses memset for memory clearing operations
- Uses Trace for logging (Verbose for success, Error for failure)

### Performance Considerations
- Time complexity: O(n) where n = total buffer size in bytes
- Memory operations: Two memset calls (buffer data + metadata structure)
- Fast operation: memset is highly optimized for bulk memory operations

### Unittests
 - ClearsAllElements : verify all buffer positions are zeroed after Clear
 - ResetsElementCount : verify elementCount is reset to 0 after Clear
 - ResetsAllMetadata : verify all metadata fields (elementCount, capacity, etc.) are zeroed
 - ReturnsTrue : verify Clear returns TRUE when buffer is initialized
 - ClearEmptyBuffer : verify clearing an already-empty buffer returns TRUE
 - ClearAfterPush : verify Clear works correctly after pushing elements
 - ClearAfterPop : verify Clear works correctly after popping elements
 - MultipleClearCalls : verify consecutive Clear calls all return TRUE
 - ClearFullBuffer : verify Clear works when buffer is at capacity
 - ClearPartialBuffer : verify Clear works when buffer is partially filled
 - PreservesConfiguration : verify buffer configuration (capacity, elementSize) unchanged after Clear
 - CanReuseAfterClear : verify buffer can be reused (push/pop) immediately after Clear
*)
Clear := FALSE;
IF isInitialized THEN
	// Clear the local buffer
	memset(pBuffer.pValue, 16#0, TO_UDINT(pBuffer.diSize));
	memset(ADR(BufferMetadata), 16#0, SIZEOF(BufferMetadata));

	// after bufferMetadata clear re-set capacity
	bufferMetadata.capacity := bufferConfiguration.capacity;
	Clear					:= TRUE;
ELSE
	Trace.Error(__POUNAME(), 'Buffer was not properly initialized before clearing buffer');
END_IF

IF Clear THEN
	Trace.Verbose(__POUNAME(), 'executed');
ELSE
	Trace.Error(__POUNAME(), 'FAILED');
END_IF
END_METHOD

PROPERTY Configuration : REFERENCE TO ST_BufferConfiguration
GET
Configuration REF= bufferConfiguration;
END_GET
END_PROPERTY

METHOD PRIVATE CountDecrement
// Decrement element count, increment capacity
bufferMetadata.elementCount := bufferMetadata.elementCount - 1;
bufferMetadata.capacity		:= bufferMetadata.capacity + 1;
END_METHOD

METHOD PRIVATE CountIncrement
// Increment element count, decrement capacity
bufferMetadata.elementCount := bufferMetadata.elementCount + 1;
bufferMetadata.capacity		:= bufferMetadata.capacity - 1;
END_METHOD

// Deletes element at specified index position, BUT DOES NOT SHIFT
METHOD DeleteAtIndex : BOOL
VAR_INPUT
	index : DINT;
END_VAR

VAR
	offset		 : DINT;
	destAddr	 : PVOID;
	srcAddr		 : PVOID;
	nBytes		 : UDINT;
	rebasedIndex : DINT;
END_VAR

(*
## Detailed Description

Deletes the element at the specified index position by zeroing out its memory location.
This is a low-level primitive operation that clears data in place without shifting other
elements or modifying metadata counters. The caller is responsible for managing element
count and buffer state if needed.

### Operation Sequence
1. Validates that index is within valid range [0, capacity)
2. Calculates byte offset to the target element position
3. Clears the element data using memset (sets all bytes to 0x00)
4. Returns TRUE on successful deletion

### Key Features
- **Low-level primitive**: Does NOT modify metadata counters - caller's responsibility
- **No state checking**: Does NOT validate if position is filled or if buffer is empty
- **Direct deletion**: Clears data at specific index WITHOUT shifting elements
- **Bounds checking**: Validates index against capacity only (not elementCount)
- **Memory safety**: Prevents deletion at invalid indices
- **Error logging**: Traces error with index value when deletion fails

### Usage Example
```iecst
VAR
    buffer : AnyBuffer(pBuffer := myArray, bufferBoundLower := 0, bufferBoundUpper := 9, isBufferPersistent := FALSE);
    success : BOOL;
END_VAR

// Delete element at index 3 (caller must manage elementCount)
success := buffer.DeleteAtIndex(3);
IF success THEN
    // Element at index 3 is now zeroed
    // NOTE: elementCount is NOT changed - caller must decrement if needed
END_IF
```

### Important Notes
- **No metadata changes**: Does NOT modify elementCount or any other metadata
- **Caller responsibility**: Calling code must manage element count if required
- **No shifting**: Does NOT shift remaining elements to fill the gap
- **No state checking**: Works regardless of whether position is filled or buffer is empty
- **Index range**: Valid indices are [0, capacity-1], not [0, elementCount-1]
- **Internal use**: Primarily used internally by PopLeft, PopRight, and PopAtIndex

### Return Value
- **TRUE**: Element was successfully deleted (zeroed at specified index)
- **FALSE**: Deletion failed due to invalid index (out of bounds)

### Error Conditions
- Returns FALSE and logs error if index < 0
- Returns FALSE and logs error if index >= capacity
- Error message includes the invalid index value for debugging

### Side Effects
- Zeros out all bytes of the element at the specified index
- **Does NOT** modify bufferMetadata.elementCount
- **Does NOT** modify any other element positions
- **Does NOT** shift elements to maintain contiguity
- **Does NOT** check if position was filled before deletion

### Dependencies
- Uses memset for memory clearing operation
- Uses Trace for error logging
- Requires valid buffer configuration (capacity, elementSize)

### Performance Considerations
- Time complexity: O(1) - constant time operation
- Memory operations: Single memset call for one element
- Fast operation: No element shifting, no metadata updates, no state checking

### Comparison with Other Methods
- **DeleteAtIndex**: Clears in place, no metadata change (O(1))
- **PopAtIndex**: Clears, shifts elements, updates count (O(n))
- **PopLeft/PopRight**: Specialized pop with shifting and count update (O(n))

### Unittests
 - DeletesAtValidIndex : verify element at valid index is zeroed after deletion
 - ReturnsTrueOnSuccess : verify method returns TRUE when deletion succeeds
 - ReturnsFalseOnInvalidIndex : verify method returns FALSE for out-of-bounds index
 - RejectsNegativeIndex : verify index < 0 is rejected with error log
 - RejectsIndexAtCapacity : verify index == capacity is rejected with error log
 - RejectsIndexAboveCapacity : verify index > capacity is rejected with error log
 - ExtremeBounds : verify rejection of extreme values like -10000 and very large positive indices
 - DeleteAtZero : verify deletion at first position (index 0) works correctly
 - DeleteAtCapacityMinusOne : verify deletion at last position (capacity-1) works correctly
 - DeleteAllPositions : verify deletion works correctly at all valid indices (0 through capacity-1)
 - PreservesOtherData : verify deletion at one index does not affect data at other indices
 - DeleteAlreadyEmpty : verify deleting an already-cleared position returns TRUE and remains zero
 - DeleteDoesNotShift : verify elements after deleted index remain at their original positions
 - DeleteWhenEmpty : verify deletion succeeds even when elementCount is 0 (clears position only)
 - MetadataUnchanged : verify elementCount and all metadata remain unchanged after deletion
 - ConsecutiveDeletesSamePosition : verify multiple deletes at same position succeed without metadata changes
*)
DeleteAtIndex := FALSE;
// check index
IF index < bufferConfiguration.bufferBoundLower OR index > bufferConfiguration.bufferBoundUpper THEN
	Trace.Error(__POUNAME(), CONCAT('Delete attempt at invalid index ', TO_STRING(index)));
	RETURN;
END_IF;

// rebasedIndex necessary if LL <> 0
rebasedIndex := index - bufferConfiguration.bufferBoundLower;

// Delete index element data
offset	 := rebasedIndex * bufferConfiguration.elementSize;
destAddr := ADR(pBuffer.pValue[offset]);
nBytes	 := TO_UDINT(bufferConfiguration.elementSize);
memset(destAddr, 16#0, nBytes);
DeleteAtIndex := TRUE;
END_METHOD

//FB_Exit must be implemented explicitly. If there is an implementation, then the

//method is called before the controller removes the code of the function block instance

//(implicit call). The return value is not evaluated.
METHOD FB_Exit : BOOL
VAR_INPUT
	bInCopyCode : BOOL; // TRUE: the exit method is called in order to leave the instance which will be copied afterwards (online change).  
END_VAR
__DELETE(pBufferTemp); // Delete if any exist
END_METHOD

//FB_Init is always available implicitly and it is used primarily for initialization.

//The return value is not evaluated. For a specific influence, you can also declare the

//methods explicitly and provide additional code there with the standard initialization

//code. You can evaluate the return value.
METHOD FB_Init : BOOL
VAR_INPUT
	bInitRetains	   : BOOL; // TRUE: the retain variables are initialized (reset warm / reset cold)
	bInCopyCode		   : BOOL; // TRUE: the instance will be copied to the copy code afterward (online change)   
	pBuffer			   : ANY;  // ANY to the buffer	
	bufferBoundLower   : DINT; // Lower boundary of the buffer
	bufferBoundUpper   : DINT; // Upper boundary of the buffer
	isBufferPersistent : BOOL; // Does the buffer need to be in persistent data?
END_VAR
THIS^.bufferConfiguration.isPersistent := isBufferPersistent;
// use the initialization method

// Valid pointer & strategy
IF pBuffer.pValue <> 0 THEN // AND_THEN
	//	bufferBoundLower = 0 			THEN
	THIS^.pBuffer						 := pBuffer;
	bufferConfiguration.bufferBoundLower := bufferBoundLower;
	bufferConfiguration.bufferBoundUpper := bufferBoundUpper;
	bufferConfiguration.capacity		 := bufferBoundUpper - bufferBoundLower + 1;
	IF NOT isBufferPersistent THEN
		// Clear the local buffer
		//memset(pBuffer.pValue, 16#0, TO_UDINT(pBuffer.diSize));
		memset(ADR(BufferMetadata), 16#0, SIZEOF(BufferMetadata));
	END_IF

	// At least 1 element? Is it an array?   	
	IF bufferConfiguration.capacity < 1 THEN
		// DO NOT USE TRACE IN THE FB_INIT METHODS
		// Trace.Error(__POUNAME(), 'Number of buffer elements < 1');
		bufferConfiguration.capacity := 0;
		isInitialized				 := FALSE;
	ELSE
		bufferConfiguration.elementSize := pBuffer.diSize / bufferConfiguration.capacity;
		bufferConfiguration.bufferSize	:= bufferConfiguration.capacity * bufferConfiguration.elementSize;
		IF NOT isBufferPersistent THEN
			// after bufferMetadata clear re-set capacity
			bufferMetadata.capacity := bufferConfiguration.capacity;
		END_IF

		// Temp buffer for the element
		pBufferTemp	  := __NEW(BYTE, TO_UDINT(bufferConfiguration.elementSize));
		isInitialized := TRUE;
	END_IF
END_IF
END_METHOD

METHOD FB_Reinit : BOOL
IF bufferConfiguration.elementSize > 0 THEN
	pBufferTemp := __NEW(BYTE, TO_UDINT(bufferConfiguration.elementSize));
END_IF
END_METHOD

PROPERTY isEmpty : BOOL
GET
isEmpty := (metaData.capacity >= bufferConfiguration.capacity);
END_GET
END_PROPERTY

PROPERTY isFull : BOOL
GET
isFull := (metaData.capacity <= 0);
END_GET
END_PROPERTY

PROPERTY Metadata : REFERENCE TO ST_BufferMetadata
GET
Metadata REF= bufferMetadata;
END_GET
END_PROPERTY

// Retrieve an element at a specific index without removing it from the buffer
METHOD PeekAtIndex : BOOL
VAR_INPUT
	index	: DINT;
	element : ANY;
END_VAR

VAR
	offset		 : DINT;
	destAddr	 : PVOID;
	srcAddr		 : PVOID;
	nBytes		 : UDINT;
	rebasedIndex : DINT;
END_VAR

(*
## Detailed Description

Retrieves an element at the specified index from the buffer without removing it or
modifying the buffer in any way. This is a read-only operation that provides random-access
read capability for the buffer. The buffer remains unchanged after this operation - no
elements are removed, shifted, or modified, and the element count stays the same.

### Operation Sequence
1. Validates that index is within valid range (0 to elementCount-1)
2. Validates that element size matches buffer element size (if element.diSize > 0)
3. Copies the element at the specified index to the output parameter
4. Returns without modifying the buffer

### Use Cases
```iecst
VAR
    buffer : AnyBuffer;
    value : DINT;
END_VAR

// Peek at elements without removing them
buffer.PushRight(100);  // [100]
buffer.PushRight(200);  // [100, 200]
buffer.PushRight(300);  // [100, 200, 300]

buffer.PeekAtIndex(0, value);  // value = 100, buffer still [100, 200, 300]
buffer.PeekAtIndex(1, value);  // value = 200, buffer still [100, 200, 300]
buffer.PeekAtIndex(2, value);  // value = 300, buffer still [100, 200, 300]

// Buffer unchanged - still contains all 3 elements
```

### Performance Considerations
- **Time complexity**: O(1) - constant time operation (direct indexed access)
- **Memory operations**: Single memcpy for element retrieval only
- **No buffer modifications**: No shifting, clearing, or count changes
- **Read-only**: Safe to call multiple times on same index
- Optimal for inspecting buffer contents without consumption
- Use for lookahead, validation, or monitoring buffer state

### Return Value
- **TRUE**: Element was successfully retrieved from the specified index
- **FALSE**: Peek operation failed (see error conditions)

### Error Conditions
- Returns FALSE and logs error if index is out of bounds (< 0 or >= elementCount)
- Returns FALSE and logs error if buffer is empty (elementCount = 0)
- Returns FALSE and logs error if element size doesn't match buffer element size (when element.diSize > 0)
- Element parameter can have diSize = 0 to skip copying (returns TRUE if index valid)

### Side Effects
- **None** - This is a read-only operation with no side effects
- Buffer contents remain unchanged
- Element count remains unchanged
- No elements are moved, cleared, or modified

### Dependencies
- Uses memcpy for element retrieval
- Uses Trace for error logging

### Comparison with Other Methods
- **PeekAtIndex**: Read element at any index - O(1), no modifications
- **PopAtIndex**: Read and remove element at any index - O(n), modifies buffer
- **PopLeft**: Read and remove first element - O(n), modifies buffer
- **PopRight**: Read and remove last element - O(1), modifies buffer
- **GetAtIndex** (if exists): Similar read-only operation

### Unittests
 - PeekFromBeginning : verify peeking at index 0 retrieves first element without modification
 - PeekFromMiddle : verify peeking from middle index retrieves correct element
 - PeekFromEnd : verify peeking at last index retrieves last element
 - ReturnsTrueOnSuccess : verify method returns TRUE when peek succeeds
 - ReturnsFalseOnNegativeIndex : verify FALSE returned for negative index
 - ReturnsFalseOnIndexOutOfBounds : verify FALSE returned when index >= elementCount
 - ReturnsFalseOnEmptyBuffer : verify FALSE returned when buffer is empty (elementCount = 0)
 - WrongElementSize : verify FALSE returned when element size doesn't match
 - EmptyElement : verify behavior when element.diSize is 0 (validation only, no copy)
 - BufferUnchangedAfterPeek : verify buffer contents unchanged after peek
 - ElementCountUnchanged : verify elementCount remains same after peek
 - MultiplePeeksOnSameIndex : verify can peek same index multiple times with consistent results
 - PeekAllPositions : verify can peek all valid positions in sequence
 - ElementOrderUnchanged : verify element order unchanged after multiple peeks
 - ConsecutivePeeks : verify multiple consecutive peeks at different indices work correctly
*)
PeekAtIndex := FALSE;
// Check index bounds, can peek every position even when not filled in
IF index < bufferConfiguration.bufferBoundLower OR index > bufferConfiguration.bufferBoundUpper THEN
	Trace.Error(__POUNAME(), CONCAT('Peek attempt at invalid index ', TO_STRING(index)));
	RETURN;
END_IF

// Check if buffer is empty
IF isEmpty THEN
	Trace.Error(__POUNAME(), 'Peek attempt on empty buffer');
	RETURN;
END_IF

// Check element size if copy is requested (element.diSize > 0)
IF element.diSize <> bufferConfiguration.elementSize THEN
	Trace.Error(__POUNAME(), CONCAT('Element size mismatch: expected ', CONCAT(TO_STRING(bufferConfiguration.elementSize), CONCAT(', got ', TO_STRING(element.diSize)))));
	RETURN;
END_IF

// rebasedIndex necessary if LL <> 0
rebasedIndex := index - bufferConfiguration.bufferBoundLower;

// Copy element at index to output parameter (if element.diSize > 0)
offset	 := rebasedIndex * bufferConfiguration.elementSize;
destAddr := element.pValue;
srcAddr	 := ADR(pBuffer.pValue[offset]);
nBytes	 := TO_UDINT(element.diSize);
memcpy(destAddr, srcAddr, nBytes);

// No buffer modifications - read-only operation
PeekAtIndex := TRUE;
END_METHOD

// Remove and retrieve an element at a specific index, decrement the element counter and shift remaining elements left
METHOD PopAtIndex : BOOL
VAR_INPUT
	index	   : DINT;
	element	   : ANY;
	popDiscard : BOOL := FALSE; // When TRUE, element is removed but not copied (type checking skipped)
END_VAR

VAR
	offset			: DINT;
	destAddr		: PVOID;
	srcAddr			: PVOID;
	nBytes			: UDINT;
	elementsToShift : DINT;
	rebasedIndex	: DINT;
END_VAR

(*
## Detailed Description

Removes an element at the specified index from the buffer and optionally copies it to
the provided element parameter. All elements after the removed index are shifted one
position to the left to maintain contiguous storage. This provides random-access pop
capability for the buffer, allowing removal from any position.

### Operation Sequence
1. Validates that index is within valid range (0 to elementCount-1)
2. Validates that element size matches buffer element size (if element.diSize > 0)
3. Copies the element at the specified index to the output parameter
4. Shifts all elements after the index one position to the left using MEMMOVE
5. Clears the last position (now empty after the shift)
6. Decrements the element count

### Use Cases
```iecst
VAR
    buffer : AnyBuffer;
    value : DINT;
END_VAR

// Remove element from middle of buffer
buffer.PushRight(100);  // [100]
buffer.PushRight(200);  // [100, 200]
buffer.PushRight(300);  // [100, 200, 300]
buffer.PopAtIndex(1, value);  // value = 200, buffer = [100, 300]
```

### Performance Considerations
- **Time complexity**: O(n) - requires shifting elements after the index
- **Memory operations**: One memcpy for retrieval, one MEMMOVE for shifting, one memset for clearing
- **Cost varies by index**:
  - PopAtIndex(0) is equivalent to PopLeft - shifts all remaining elements
  - PopAtIndex(elementCount-1) is equivalent to PopRight - no shifting needed
  - Middle indices require partial shifting
- Use PopRight for O(1) removal when index doesn't matter
- Use for priority queues or sorted list maintenance

### Return Value
- **TRUE**: Element was successfully popped from the specified index
- **FALSE**: Pop operation failed (see error conditions)

### Error Conditions
- Returns FALSE and logs error if index is out of bounds (< 0 or >= elementCount)
- Returns FALSE and logs error if buffer is empty (elementCount = 0)
- Returns FALSE and logs error if element size doesn't match buffer element size (when element.diSize > 0)
- Element parameter can have diSize = 0 to discard the value without copying

### Side Effects
- Shifts all elements after the index one position to the left
- Clears the last element position (sets to zero)
- Decrements bufferMetadata.elementCount by 1

### Dependencies
- Uses memcpy for element retrieval
- Uses MEMMOVE for shifting elements (handles overlapping memory)
- Uses memset for clearing the last position
- Uses Trace for error logging

### Comparison with Other Methods
- **PopAtIndex(0)**: Same as PopLeft - removes from front, shifts all - O(n)
- **PopAtIndex(elementCount-1)**: Same as PopRight - removes from back, no shift - O(1)
- **PopAtIndex(middle)**: Removes from middle, shifts elements after index - O(n)
- **DeleteAtIndex**: Removes without retrieving value - O(1) for last index, O(n) otherwise

